//     PlcTask Inputs/MAIN.force_rb_X[146] <-> Status process data mapping/force_rb_X
//     PlcTask Inputs/MAIN.force_rb_Y[146] <-> Status process data mapping/force_rb_Y
//     PlcTask Inputs/MAIN.force_rb_Z[146] <-> Status process data mapping/force_rb_Z
//     PlcTask Inputs/MAIN.force_sp_X[146] <-> Status process data mapping/force_sp_X
//     PlcTask Inputs/MAIN.force_sp_Y[146] <-> Status process data mapping/force_sp_Y
//     PlcTask Inputs/MAIN.force_sp_Z[146] <-> Status process data mapping/force_sp_Z
//     PlcTask Inputs/MAIN.pwm1[146] <-> Status process data mapping/pwm1
//     PlcTask Inputs/MAIN.pwm2[146] <-> Status process data mapping/pwm2
//     PlcTask Inputs/MAIN.pwm3[146] <-> Status process data mapping/pwm3
//     PlcTask Outputs/MAIN.enable_cmd[146] <-> Control process data mapping/enable
//     PlcTask Outputs/MAIN.force_cmd_X[146] <-> Control process data mapping/force_sp_X
//     PlcTask Outputs/MAIN.force_cmd_Y[146] <-> Control process data mapping/force_sp_Y
//     PlcTask Outputs/MAIN.force_cmd_Z[146] <-> Control process data mapping/force_sp_Z
//     PlcTask Outputs/MAIN.msthb[156] <-> Control process data mapping/msthb
//   SAsetGains/SAsetGains Instance <-> Device 1 (EtherCAT)/Box 148 (m1eph)/Box 157 (m1sa)
//     PlcTask Inputs/MAIN.cloop_stat[147] <-> Status process data mapping/close_loop
//     PlcTask Inputs/MAIN.enable_stat[147] <-> Status process data mapping/enable
//     PlcTask Inputs/MAIN.force_rb_X[147] <-> Status process data mapping/force_rb_X
//     PlcTask Inputs/MAIN.force_rb_Y[147] <-> Status process data mapping/force_rb_Y
//     PlcTask Inputs/MAIN.force_rb_Z[147] <-> Status process data mapping/force_rb_Z
//     PlcTask Inputs/MAIN.force_sp_X[147] <-> Status process data mapping/force_sp_X
//     PlcTask Inputs/MAIN.force_sp_Y[147] <-> Status process data mapping/force_sp_Y
//     PlcTask Inputs/MAIN.force_sp_Z[147] <-> Status process data mapping/force_sp_Z
//     PlcTask Inputs/MAIN.pwm1[147] <-> Status process data mapping/pwm1
//     PlcTask Inputs/MAIN.pwm2[147] <-> Status process data mapping/pwm2
//     PlcTask Inputs/MAIN.pwm3[147] <-> Status process data mapping/pwm3
//     PlcTask Outputs/MAIN.enable_cmd[147] <-> Control process data mapping/enable
//     PlcTask Outputs/MAIN.force_cmd_X[147] <-> Control process data mapping/force_sp_X
//     PlcTask Outputs/MAIN.force_cmd_Y[147] <-> Control process data mapping/force_sp_Y
//     PlcTask Outputs/MAIN.force_cmd_Z[147] <-> Control process data mapping/force_sp_Z
//     PlcTask Outputs/MAIN.msthb[157] <-> Control process data mapping/msthb
//   SAsetGains/SAsetGains Instance <-> Device 1 (EtherCAT)/Box 148 (m1eph)/Box 158 (m1sa)
//     PlcTask Inputs/MAIN.cloop_stat[148] <-> Status process data mapping/close_loop
//     PlcTask Inputs/MAIN.enable_stat[148] <-> Status process data mapping/enable
//     PlcTask Inputs/MAIN.force_rb_X[148] <-> Status process data mapping/force_rb_X
//     PlcTask Inputs/MAIN.force_rb_Y[148] <-> Status process data mapping/force_rb_Y
//     PlcTask Inputs/MAIN.force_rb_Z[148] <-> Status process data mapping/force_rb_Z
//     PlcTask Inputs/MAIN.force_sp_X[148] <-> Status process data mapping/force_sp_X
//     PlcTask Inputs/MAIN.force_sp_Y[148] <-> Status process data mapping/force_sp_Y
//     PlcTask Inputs/MAIN.force_sp_Z[148] <-> Status process data mapping/force_sp_Z
//     PlcTask Inputs/MAIN.pwm1[148] <-> Status process data mapping/pwm1
//     PlcTask Inputs/MAIN.pwm2[148] <-> Status process data mapping/pwm2
//     PlcTask Inputs/MAIN.pwm3[148] <-> Status process data mapping/pwm3
//     PlcTask Outputs/MAIN.enable_cmd[148] <-> Control process data mapping/enable
//     PlcTask Outputs/MAIN.force_cmd_X[148] <-> Control process data mapping/force_sp_X
//     PlcTask Outputs/MAIN.force_cmd_Y[148] <-> Control process data mapping/force_sp_Y
//     PlcTask Outputs/MAIN.force_cmd_Z[148] <-> Control process data mapping/force_sp_Z
//     PlcTask Outputs/MAIN.msthb[158] <-> Control process data mapping/msthb
//   SAsetGains/SAsetGains Instance <-> Device 1 (EtherCAT)/Box 148 (m1eph)/Box 159 (m1sa)
//     PlcTask Inputs/MAIN.cloop_stat[149] <-> Status process data mapping/close_loop
//     PlcTask Inputs/MAIN.enable_stat[149] <-> Status process data mapping/enable
//     PlcTask Inputs/MAIN.force_rb_X[149] <-> Status process data mapping/force_rb_X
//     PlcTask Inputs/MAIN.force_rb_Y[149] <-> Status process data mapping/force_rb_Y
//     PlcTask Inputs/MAIN.force_rb_Z[149] <-> Status process data mapping/force_rb_Z
//     PlcTask Inputs/MAIN.force_sp_X[149] <-> Status process data mapping/force_sp_X
//     PlcTask Inputs/MAIN.force_sp_Y[149] <-> Status process data mapping/force_sp_Y
//     PlcTask Inputs/MAIN.force_sp_Z[149] <-> Status process data mapping/force_sp_Z
//     PlcTask Inputs/MAIN.pwm1[149] <-> Status process data mapping/pwm1
//     PlcTask Inputs/MAIN.pwm2[149] <-> Status process data mapping/pwm2
//     PlcTask Inputs/MAIN.pwm3[149] <-> Status process data mapping/pwm3
//     PlcTask Outputs/MAIN.enable_cmd[149] <-> Control process data mapping/enable
//     PlcTask Outputs/MAIN.force_cmd_X[149] <-> Control process data mapping/force_sp_X
//     PlcTask Outputs/MAIN.force_cmd_Y[149] <-> Control process data mapping/force_sp_Y
//     PlcTask Outputs/MAIN.force_cmd_Z[149] <-> Control process data mapping/force_sp_Z
//     PlcTask Outputs/MAIN.msthb[159] <-> Control process data mapping/msthb
//   SAsetGains/SAsetGains Instance <-> Device 1 (EtherCAT)/Box 148 (m1eph)/Box 160 (m1sa)
//     PlcTask Inputs/MAIN.cloop_stat[150] <-> Status process data mapping/close_loop
//     PlcTask Inputs/MAIN.enable_stat[150] <-> Status process data mapping/enable
//     PlcTask Inputs/MAIN.force_rb_X[150] <-> Status process data mapping/force_rb_X
//     PlcTask Inputs/MAIN.force_rb_Y[150] <-> Status process data mapping/force_rb_Y
//     PlcTask Inputs/MAIN.force_rb_Z[150] <-> Status process data mapping/force_rb_Z
//     PlcTask Inputs/MAIN.force_sp_X[150] <-> Status process data mapping/force_sp_X
//     PlcTask Inputs/MAIN.force_sp_Y[150] <-> Status process data mapping/force_sp_Y
//     PlcTask Inputs/MAIN.force_sp_Z[150] <-> Status process data mapping/force_sp_Z
//     PlcTask Inputs/MAIN.pwm1[150] <-> Status process data mapping/pwm1
//     PlcTask Inputs/MAIN.pwm2[150] <-> Status process data mapping/pwm2
//     PlcTask Inputs/MAIN.pwm3[150] <-> Status process data mapping/pwm3
//     PlcTask Outputs/MAIN.enable_cmd[150] <-> Control process data mapping/enable
//     PlcTask Outputs/MAIN.force_cmd_X[150] <-> Control process data mapping/force_sp_X
//     PlcTask Outputs/MAIN.force_cmd_Y[150] <-> Control process data mapping/force_sp_Y
//     PlcTask Outputs/MAIN.force_cmd_Z[150] <-> Control process data mapping/force_sp_Z
//     PlcTask Outputs/MAIN.msthb[160] <-> Control process data mapping/msthb
//   SAsetGains/SAsetGains Instance <-> Device 1 (EtherCAT)/Box 148 (m1eph)/Box 161 (m1sa)
//     PlcTask Inputs/MAIN.cloop_stat[151] <-> Status process data mapping/close_loop
//     PlcTask Inputs/MAIN.enable_stat[151] <-> Status process data mapping/enable
//     PlcTask Inputs/MAIN.force_rb_X[151] <-> Status process data mapping/force_rb_X
//     PlcTask Inputs/MAIN.force_rb_Y[151] <-> Status process data mapping/force_rb_Y
//     PlcTask Inputs/MAIN.force_rb_Z[151] <-> Status process data mapping/force_rb_Z
//     PlcTask Inputs/MAIN.force_sp_X[151] <-> Status process data mapping/force_sp_X
//     PlcTask Inputs/MAIN.force_sp_Y[151] <-> Status process data mapping/force_sp_Y
//     PlcTask Inputs/MAIN.force_sp_Z[151] <-> Status process data mapping/force_sp_Z
//     PlcTask Inputs/MAIN.pwm1[151] <-> Status process data mapping/pwm1
//     PlcTask Inputs/MAIN.pwm2[151] <-> Status process data mapping/pwm2
//     PlcTask Inputs/MAIN.pwm3[151] <-> Status process data mapping/pwm3
//     PlcTask Outputs/MAIN.enable_cmd[151] <-> Control process data mapping/enable
//     PlcTask Outputs/MAIN.force_cmd_X[151] <-> Control process data mapping/force_sp_X
//     PlcTask Outputs/MAIN.force_cmd_Y[151] <-> Control process data mapping/force_sp_Y
//     PlcTask Outputs/MAIN.force_cmd_Z[151] <-> Control process data mapping/force_sp_Z
//     PlcTask Outputs/MAIN.msthb[161] <-> Control process data mapping/msthb
//   SAsetGains/SAsetGains Instance <-> Device 1 (EtherCAT)/Box 148 (m1eph)/Box 162 (m1sa)
//     PlcTask Inputs/MAIN.cloop_stat[152] <-> Status process data mapping/close_loop
//     PlcTask Inputs/MAIN.enable_stat[152] <-> Status process data mapping/enable
//     PlcTask Inputs/MAIN.force_rb_X[152] <-> Status process data mapping/force_rb_X
//     PlcTask Inputs/MAIN.force_rb_Y[152] <-> Status process data mapping/force_rb_Y
//     PlcTask Inputs/MAIN.force_rb_Z[152] <-> Status process data mapping/force_rb_Z
//     PlcTask Inputs/MAIN.force_sp_X[152] <-> Status process data mapping/force_sp_X
//     PlcTask Inputs/MAIN.force_sp_Y[152] <-> Status process data mapping/force_sp_Y
//     PlcTask Inputs/MAIN.force_sp_Z[152] <-> Status process data mapping/force_sp_Z
//     PlcTask Inputs/MAIN.pwm1[152] <-> Status process data mapping/pwm1
//     PlcTask Inputs/MAIN.pwm2[152] <-> Status process data mapping/pwm2
//     PlcTask Inputs/MAIN.pwm3[152] <-> Status process data mapping/pwm3
//     PlcTask Outputs/MAIN.enable_cmd[152] <-> Control process data mapping/enable
//     PlcTask Outputs/MAIN.force_cmd_X[152] <-> Control process data mapping/force_sp_X
//     PlcTask Outputs/MAIN.force_cmd_Y[152] <-> Control process data mapping/force_sp_Y
//     PlcTask Outputs/MAIN.force_cmd_Z[152] <-> Control process data mapping/force_sp_Z
//     PlcTask Outputs/MAIN.msthb[162] <-> Control process data mapping/msthb
//   SAsetGains/SAsetGains Instance <-> Device 1 (EtherCAT)/Box 148 (m1eph)/Box 163 (m1sa)
//     PlcTask Inputs/MAIN.cloop_stat[153] <-> Status process data mapping/close_loop
//     PlcTask Inputs/MAIN.enable_stat[153] <-> Status process data mapping/enable
//     PlcTask Inputs/MAIN.force_rb_X[153] <-> Status process data mapping/force_rb_X
//     PlcTask Inputs/MAIN.force_rb_Y[153] <-> Status process data mapping/force_rb_Y
//     PlcTask Inputs/MAIN.force_rb_Z[153] <-> Status process data mapping/force_rb_Z
//     PlcTask Inputs/MAIN.force_sp_X[153] <-> Status process data mapping/force_sp_X
//     PlcTask Inputs/MAIN.force_sp_Y[153] <-> Status process data mapping/force_sp_Y
//     PlcTask Inputs/MAIN.force_sp_Z[153] <-> Status process data mapping/force_sp_Z
//     PlcTask Inputs/MAIN.pwm1[153] <-> Status process data mapping/pwm1
//     PlcTask Inputs/MAIN.pwm2[153] <-> Status process data mapping/pwm2
//     PlcTask Inputs/MAIN.pwm3[153] <-> Status process data mapping/pwm3
//     PlcTask Outputs/MAIN.enable_cmd[153] <-> Control process data mapping/enable
//     PlcTask Outputs/MAIN.force_cmd_X[153] <-> Control process data mapping/force_sp_X
//     PlcTask Outputs/MAIN.force_cmd_Y[153] <-> Control process data mapping/force_sp_Y
//     PlcTask Outputs/MAIN.force_cmd_Z[153] <-> Control process data mapping/force_sp_Z
//     PlcTask Outputs/MAIN.msthb[163] <-> Control process data mapping/msthb
//   SAsetGains/SAsetGains Instance <-> Device 1 (EtherCAT)/Box 148 (m1eph)/Box 164 (m1sa)
//     PlcTask Inputs/MAIN.cloop_stat[154] <-> Status process data mapping/close_loop
//     PlcTask Inputs/MAIN.enable_stat[154] <-> Status process data mapping/enable
//     PlcTask Inputs/MAIN.force_rb_X[154] <-> Status process data mapping/force_rb_X
//     PlcTask Inputs/MAIN.force_rb_Y[154] <-> Status process data mapping/force_rb_Y
//     PlcTask Inputs/MAIN.force_rb_Z[154] <-> Status process data mapping/force_rb_Z
//     PlcTask Inputs/MAIN.force_sp_X[154] <-> Status process data mapping/force_sp_X
//     PlcTask Inputs/MAIN.force_sp_Y[154] <-> Status process data mapping/force_sp_Y
//     PlcTask Inputs/MAIN.force_sp_Z[154] <-> Status process data mapping/force_sp_Z
//     PlcTask Inputs/MAIN.pwm1[154] <-> Status process data mapping/pwm1
//     PlcTask Inputs/MAIN.pwm2[154] <-> Status process data mapping/pwm2
//     PlcTask Inputs/MAIN.pwm3[154] <-> Status process data mapping/pwm3
//     PlcTask Outputs/MAIN.enable_cmd[154] <-> Control process data mapping/enable
//     PlcTask Outputs/MAIN.force_cmd_X[154] <-> Control process data mapping/force_sp_X
//     PlcTask Outputs/MAIN.force_cmd_Y[154] <-> Control process data mapping/force_sp_Y
//     PlcTask Outputs/MAIN.force_cmd_Z[154] <-> Control process data mapping/force_sp_Z
//     PlcTask Outputs/MAIN.msthb[164] <-> Control process data mapping/msthb
//   SAsetGains/SAsetGains Instance <-> Device 1 (EtherCAT)/Box 165 (m1eph)
//     PlcTask Outputs/MAIN.msthb[165] <-> Control process data mapping/msthb
//   SAsetGains/SAsetGains Instance <-> Device 1 (EtherCAT)/Box 165 (m1eph)/Box 166 (m1sa)
//     PlcTask Inputs/MAIN.cloop_stat[155] <-> Status process data mapping/close_loop
//     PlcTask Inputs/MAIN.enable_stat[155] <-> Status process data mapping/enable
//     PlcTask Inputs/MAIN.force_rb_X[155] <-> Status process data mapping/force_rb_X
//     PlcTask Inputs/MAIN.force_rb_Y[155] <-> Status process data mapping/force_rb_Y
//     PlcTask Inputs/MAIN.force_rb_Z[155] <-> Status process data mapping/force_rb_Z
//     PlcTask Inputs/MAIN.force_sp_X[155] <-> Status process data mapping/force_sp_X
//     PlcTask Inputs/MAIN.force_sp_Y[155] <-> Status process data mapping/force_sp_Y
//     PlcTask Inputs/MAIN.force_sp_Z[155] <-> Status process data mapping/force_sp_Z
//     PlcTask Inputs/MAIN.pwm1[155] <-> Status process data mapping/pwm1
//     PlcTask Inputs/MAIN.pwm2[155] <-> Status process data mapping/pwm2
//     PlcTask Inputs/MAIN.pwm3[155] <-> Status process data mapping/pwm3
//     PlcTask Outputs/MAIN.enable_cmd[155] <-> Control process data mapping/enable
//     PlcTask Outputs/MAIN.force_cmd_X[155] <-> Control process data mapping/force_sp_X
//     PlcTask Outputs/MAIN.force_cmd_Y[155] <-> Control process data mapping/force_sp_Y
//     PlcTask Outputs/MAIN.force_cmd_Z[155] <-> Control process data mapping/force_sp_Z
//     PlcTask Outputs/MAIN.msthb[166] <-> Control process data mapping/msthb
//   SAsetGains/SAsetGains Instance <-> Device 1 (EtherCAT)/Box 165 (m1eph)/Box 167 (m1sa)
//     PlcTask Inputs/MAIN.cloop_stat[156] <-> Status process data mapping/close_loop
//     PlcTask Inputs/MAIN.enable_stat[156] <-> Status process data mapping/enable
//     PlcTask Inputs/MAIN.force_rb_X[156] <-> Status process data mapping/force_rb_X
//     PlcTask Inputs/MAIN.force_rb_Y[156] <-> Status process data mapping/force_rb_Y
//     PlcTask Inputs/MAIN.force_rb_Z[156] <-> Status process data mapping/force_rb_Z
//     PlcTask Inputs/MAIN.force_sp_X[156] <-> Status process data mapping/force_sp_X
//     PlcTask Inputs/MAIN.force_sp_Y[156] <-> Status process data mapping/force_sp_Y
//     PlcTask Inputs/MAIN.force_sp_Z[156] <-> Status process data mapping/force_sp_Z
//     PlcTask Inputs/MAIN.pwm1[156] <-> Status process data mapping/pwm1
//     PlcTask Inputs/MAIN.pwm2[156] <-> Status process data mapping/pwm2
//     PlcTask Inputs/MAIN.pwm3[156] <-> Status process data mapping/pwm3
//     PlcTask Outputs/MAIN.enable_cmd[156] <-> Control process data mapping/enable
//     PlcTask Outputs/MAIN.force_cmd_X[156] <-> Control process data mapping/force_sp_X
//     PlcTask Outputs/MAIN.force_cmd_Y[156] <-> Control process data mapping/force_sp_Y
//     PlcTask Outputs/MAIN.force_cmd_Z[156] <-> Control process data mapping/force_sp_Z
//     PlcTask Outputs/MAIN.msthb[167] <-> Control process data mapping/msthb
//   SAsetGains/SAsetGains Instance <-> Device 1 (EtherCAT)/Box 165 (m1eph)/Box 168 (m1sa)
//     PlcTask Inputs/MAIN.cloop_stat[157] <-> Status process data mapping/close_loop
//     PlcTask Inputs/MAIN.enable_stat[157] <-> Status process data mapping/enable
//     PlcTask Inputs/MAIN.force_rb_X[157] <-> Status process data mapping/force_rb_X
//     PlcTask Inputs/MAIN.force_rb_Y[157] <-> Status process data mapping/force_rb_Y
//     PlcTask Inputs/MAIN.force_rb_Z[157] <-> Status process data mapping/force_rb_Z
//     PlcTask Inputs/MAIN.force_sp_X[157] <-> Status process data mapping/force_sp_X
//     PlcTask Inputs/MAIN.force_sp_Y[157] <-> Status process data mapping/force_sp_Y
//     PlcTask Inputs/MAIN.force_sp_Z[157] <-> Status process data mapping/force_sp_Z
//     PlcTask Inputs/MAIN.pwm1[157] <-> Status process data mapping/pwm1
//     PlcTask Inputs/MAIN.pwm2[157] <-> Status process data mapping/pwm2
//     PlcTask Inputs/MAIN.pwm3[157] <-> Status process data mapping/pwm3
//     PlcTask Outputs/MAIN.enable_cmd[157] <-> Control process data mapping/enable
//     PlcTask Outputs/MAIN.force_cmd_X[157] <-> Control process data mapping/force_sp_X
//     PlcTask Outputs/MAIN.force_cmd_Y[157] <-> Control process data mapping/force_sp_Y
//     PlcTask Outputs/MAIN.force_cmd_Z[157] <-> Control process data mapping/force_sp_Z
//     PlcTask Outputs/MAIN.msthb[168] <-> Control process data mapping/msthb
//   SAsetGains/SAsetGains Instance <-> Device 1 (EtherCAT)/Box 165 (m1eph)/Box 169 (m1sa)
//     PlcTask Inputs/MAIN.cloop_stat[158] <-> Status process data mapping/close_loop
//     PlcTask Inputs/MAIN.enable_stat[158] <-> Status process data mapping/enable
//     PlcTask Inputs/MAIN.force_rb_X[158] <-> Status process data mapping/force_rb_X
//     PlcTask Inputs/MAIN.force_rb_Y[158] <-> Status process data mapping/force_rb_Y
//     PlcTask Inputs/MAIN.force_rb_Z[158] <-> Status process data mapping/force_rb_Z
//     PlcTask Inputs/MAIN.force_sp_X[158] <-> Status process data mapping/force_sp_X
//     PlcTask Inputs/MAIN.force_sp_Y[158] <-> Status process data mapping/force_sp_Y
//     PlcTask Inputs/MAIN.force_sp_Z[158] <-> Status process data mapping/force_sp_Z
//     PlcTask Inputs/MAIN.pwm1[158] <-> Status process data mapping/pwm1
//     PlcTask Inputs/MAIN.pwm2[158] <-> Status process data mapping/pwm2
//     PlcTask Inputs/MAIN.pwm3[158] <-> Status process data mapping/pwm3
//     PlcTask Outputs/MAIN.enable_cmd[158] <-> Control process data mapping/enable
//     PlcTask Outputs/MAIN.force_cmd_X[158] <-> Control process data mapping/force_sp_X
//     PlcTask Outputs/MAIN.force_cmd_Y[158] <-> Control process data mapping/force_sp_Y
//     PlcTask Outputs/MAIN.force_cmd_Z[158] <-> Control process data mapping/force_sp_Z
//     PlcTask Outputs/MAIN.msthb[169] <-> Control process data mapping/msthb
//   SAsetGains/SAsetGains Instance <-> Device 1 (EtherCAT)/Box 165 (m1eph)/Box 170 (m1sa)
//     PlcTask Inputs/MAIN.cloop_stat[159] <-> Status process data mapping/close_loop
//     PlcTask Inputs/MAIN.enable_stat[159] <-> Status process data mapping/enable
//     PlcTask Inputs/MAIN.force_rb_X[159] <-> Status process data mapping/force_rb_X
//     PlcTask Inputs/MAIN.force_rb_Y[159] <-> Status process data mapping/force_rb_Y
//     PlcTask Inputs/MAIN.force_rb_Z[159] <-> Status process data mapping/force_rb_Z
//     PlcTask Inputs/MAIN.force_sp_X[159] <-> Status process data mapping/force_sp_X
//     PlcTask Inputs/MAIN.force_sp_Y[159] <-> Status process data mapping/force_sp_Y
//     PlcTask Inputs/MAIN.force_sp_Z[159] <-> Status process data mapping/force_sp_Z
//     PlcTask Inputs/MAIN.pwm1[159] <-> Status process data mapping/pwm1
//     PlcTask Inputs/MAIN.pwm2[159] <-> Status process data mapping/pwm2
//     PlcTask Inputs/MAIN.pwm3[159] <-> Status process data mapping/pwm3
//     PlcTask Outputs/MAIN.enable_cmd[159] <-> Control process data mapping/enable
//     PlcTask Outputs/MAIN.force_cmd_X[159] <-> Control process data mapping/force_sp_X
//     PlcTask Outputs/MAIN.force_cmd_Y[159] <-> Control process data mapping/force_sp_Y
//     PlcTask Outputs/MAIN.force_cmd_Z[159] <-> Control process data mapping/force_sp_Z
//     PlcTask Outputs/MAIN.msthb[170] <-> Control process data mapping/msthb
//   SAsetGains/SAsetGains Instance <-> Device 1 (EtherCAT)/Box 165 (m1eph)/Box 171 (m1sa)
//     PlcTask Inputs/MAIN.cloop_stat[160] <-> Status process data mapping/close_loop
//     PlcTask Inputs/MAIN.enable_stat[160] <-> Status process data mapping/enable
//     PlcTask Inputs/MAIN.force_rb_X[160] <-> Status process data mapping/force_rb_X
//     PlcTask Inputs/MAIN.force_rb_Y[160] <-> Status process data mapping/force_rb_Y
//     PlcTask Inputs/MAIN.force_rb_Z[160] <-> Status process data mapping/force_rb_Z
//     PlcTask Inputs/MAIN.force_sp_X[160] <-> Status process data mapping/force_sp_X
//     PlcTask Inputs/MAIN.force_sp_Y[160] <-> Status process data mapping/force_sp_Y
//     PlcTask Inputs/MAIN.force_sp_Z[160] <-> Status process data mapping/force_sp_Z
//     PlcTask Inputs/MAIN.pwm1[160] <-> Status process data mapping/pwm1
//     PlcTask Inputs/MAIN.pwm2[160] <-> Status process data mapping/pwm2
//     PlcTask Inputs/MAIN.pwm3[160] <-> Status process data mapping/pwm3
//     PlcTask Outputs/MAIN.enable_cmd[160] <-> Control process data mapping/enable
//     PlcTask Outputs/MAIN.force_cmd_X[160] <-> Control process data mapping/force_sp_X
//     PlcTask Outputs/MAIN.force_cmd_Y[160] <-> Control process data mapping/force_sp_Y
//     PlcTask Outputs/MAIN.force_cmd_Z[160] <-> Control process data mapping/force_sp_Z
//     PlcTask Outputs/MAIN.msthb[171] <-> Control process data mapping/msthb
//   SAsetGains/SAsetGains Instance <-> Device 1 (EtherCAT)/Box 165 (m1eph)/Box 172 (m1sa)
//     PlcTask Inputs/MAIN.cloop_stat[161] <-> Status process data mapping/close_loop
//     PlcTask Inputs/MAIN.enable_stat[161] <-> Status process data mapping/enable
//     PlcTask Inputs/MAIN.force_rb_X[161] <-> Status process data mapping/force_rb_X
//     PlcTask Inputs/MAIN.force_rb_Y[161] <-> Status process data mapping/force_rb_Y
//     PlcTask Inputs/MAIN.force_rb_Z[161] <-> Status process data mapping/force_rb_Z
//     PlcTask Inputs/MAIN.force_sp_X[161] <-> Status process data mapping/force_sp_X
//     PlcTask Inputs/MAIN.force_sp_Y[161] <-> Status process data mapping/force_sp_Y
//     PlcTask Inputs/MAIN.force_sp_Z[161] <-> Status process data mapping/force_sp_Z
//     PlcTask Inputs/MAIN.pwm1[161] <-> Status process data mapping/pwm1
//     PlcTask Inputs/MAIN.pwm2[161] <-> Status process data mapping/pwm2
//     PlcTask Inputs/MAIN.pwm3[161] <-> Status process data mapping/pwm3
//     PlcTask Outputs/MAIN.enable_cmd[161] <-> Control process data mapping/enable
//     PlcTask Outputs/MAIN.force_cmd_X[161] <-> Control process data mapping/force_sp_X
//     PlcTask Outputs/MAIN.force_cmd_Y[161] <-> Control process data mapping/force_sp_Y
//     PlcTask Outputs/MAIN.force_cmd_Z[161] <-> Control process data mapping/force_sp_Z
//     PlcTask Outputs/MAIN.msthb[172] <-> Control process data mapping/msthb
//   SAsetGains/SAsetGains Instance <-> Device 1 (EtherCAT)/Box 165 (m1eph)/Box 173 (m1sa)
//     PlcTask Inputs/MAIN.cloop_stat[162] <-> Status process data mapping/close_loop
//     PlcTask Inputs/MAIN.enable_stat[162] <-> Status process data mapping/enable
//     PlcTask Inputs/MAIN.force_rb_X[162] <-> Status process data mapping/force_rb_X
//     PlcTask Inputs/MAIN.force_rb_Y[162] <-> Status process data mapping/force_rb_Y
//     PlcTask Inputs/MAIN.force_rb_Z[162] <-> Status process data mapping/force_rb_Z
//     PlcTask Inputs/MAIN.force_sp_X[162] <-> Status process data mapping/force_sp_X
//     PlcTask Inputs/MAIN.force_sp_Y[162] <-> Status process data mapping/force_sp_Y
//     PlcTask Inputs/MAIN.force_sp_Z[162] <-> Status process data mapping/force_sp_Z
//     PlcTask Inputs/MAIN.pwm1[162] <-> Status process data mapping/pwm1
//     PlcTask Inputs/MAIN.pwm2[162] <-> Status process data mapping/pwm2
//     PlcTask Inputs/MAIN.pwm3[162] <-> Status process data mapping/pwm3
//     PlcTask Outputs/MAIN.enable_cmd[162] <-> Control process data mapping/enable
//     PlcTask Outputs/MAIN.force_cmd_X[162] <-> Control process data mapping/force_sp_X
//     PlcTask Outputs/MAIN.force_cmd_Y[162] <-> Control process data mapping/force_sp_Y
//     PlcTask Outputs/MAIN.force_cmd_Z[162] <-> Control process data mapping/force_sp_Z
//     PlcTask Outputs/MAIN.msthb[173] <-> Control process data mapping/msthb
//   SAsetGains/SAsetGains Instance <-> Device 1 (EtherCAT)/Box 165 (m1eph)/Box 174 (m1sa)
//     PlcTask Inputs/MAIN.cloop_stat[163] <-> Status process data mapping/close_loop
//     PlcTask Inputs/MAIN.enable_stat[163] <-> Status process data mapping/enable
//     PlcTask Inputs/MAIN.force_rb_X[163] <-> Status process data mapping/force_rb_X
//     PlcTask Inputs/MAIN.force_rb_Y[163] <-> Status process data mapping/force_rb_Y
//     PlcTask Inputs/MAIN.force_rb_Z[163] <-> Status process data mapping/force_rb_Z
//     PlcTask Inputs/MAIN.force_sp_X[163] <-> Status process data mapping/force_sp_X
//     PlcTask Inputs/MAIN.force_sp_Y[163] <-> Status process data mapping/force_sp_Y
//     PlcTask Inputs/MAIN.force_sp_Z[163] <-> Status process data mapping/force_sp_Z
//     PlcTask Inputs/MAIN.pwm1[163] <-> Status process data mapping/pwm1
//     PlcTask Inputs/MAIN.pwm2[163] <-> Status process data mapping/pwm2
//     PlcTask Inputs/MAIN.pwm3[163] <-> Status process data mapping/pwm3
//     PlcTask Outputs/MAIN.enable_cmd[163] <-> Control process data mapping/enable
//     PlcTask Outputs/MAIN.force_cmd_X[163] <-> Control process data mapping/force_sp_X
//     PlcTask Outputs/MAIN.force_cmd_Y[163] <-> Control process data mapping/force_sp_Y
//     PlcTask Outputs/MAIN.force_cmd_Z[163] <-> Control process data mapping/force_sp_Z
//     PlcTask Outputs/MAIN.msthb[174] <-> Control process data mapping/msthb
//   SAsetGains/SAsetGains Instance <-> Device 1 (EtherCAT)/Box 165 (m1eph)/Box 175 (m1sa)
//     PlcTask Inputs/MAIN.cloop_stat[164] <-> Status process data mapping/close_loop
//     PlcTask Inputs/MAIN.enable_stat[164] <-> Status process data mapping/enable
//     PlcTask Inputs/MAIN.force_rb_X[164] <-> Status process data mapping/force_rb_X
//     PlcTask Inputs/MAIN.force_rb_Y[164] <-> Status process data mapping/force_rb_Y
//     PlcTask Inputs/MAIN.force_rb_Z[164] <-> Status process data mapping/force_rb_Z
//     PlcTask Inputs/MAIN.force_sp_X[164] <-> Status process data mapping/force_sp_X
//     PlcTask Inputs/MAIN.force_sp_Y[164] <-> Status process data mapping/force_sp_Y
//     PlcTask Inputs/MAIN.force_sp_Z[164] <-> Status process data mapping/force_sp_Z
//     PlcTask Inputs/MAIN.pwm1[164] <-> Status process data mapping/pwm1
//     PlcTask Inputs/MAIN.pwm2[164] <-> Status process data mapping/pwm2
//     PlcTask Inputs/MAIN.pwm3[164] <-> Status process data mapping/pwm3
//     PlcTask Outputs/MAIN.enable_cmd[164] <-> Control process data mapping/enable
//     PlcTask Outputs/MAIN.force_cmd_X[164] <-> Control process data mapping/force_sp_X
//     PlcTask Outputs/MAIN.force_cmd_Y[164] <-> Control process data mapping/force_sp_Y
//     PlcTask Outputs/MAIN.force_cmd_Z[164] <-> Control process data mapping/force_sp_Z
//     PlcTask Outputs/MAIN.msthb[175] <-> Control process data mapping/msthb
//   SAsetGains/SAsetGains Instance <-> Device 1 (EtherCAT)/Box 165 (m1eph)/Box 176 (m1sa)
//     PlcTask Inputs/MAIN.cloop_stat[165] <-> Status process data mapping/close_loop
//     PlcTask Inputs/MAIN.enable_stat[165] <-> Status process data mapping/enable
//     PlcTask Inputs/MAIN.force_rb_X[165] <-> Status process data mapping/force_rb_X
//     PlcTask Inputs/MAIN.force_rb_Y[165] <-> Status process data mapping/force_rb_Y
//     PlcTask Inputs/MAIN.force_rb_Z[165] <-> Status process data mapping/force_rb_Z
//     PlcTask Inputs/MAIN.force_sp_X[165] <-> Status process data mapping/force_sp_X
//     PlcTask Inputs/MAIN.force_sp_Y[165] <-> Status process data mapping/force_sp_Y
//     PlcTask Inputs/MAIN.force_sp_Z[165] <-> Status process data mapping/force_sp_Z
//     PlcTask Inputs/MAIN.pwm1[165] <-> Status process data mapping/pwm1
//     PlcTask Inputs/MAIN.pwm2[165] <-> Status process data mapping/pwm2
//     PlcTask Inputs/MAIN.pwm3[165] <-> Status process data mapping/pwm3
//     PlcTask Outputs/MAIN.enable_cmd[165] <-> Control process data mapping/enable
//     PlcTask Outputs/MAIN.force_cmd_X[165] <-> Control process data mapping/force_sp_X
//     PlcTask Outputs/MAIN.force_cmd_Y[165] <-> Control process data mapping/force_sp_Y
//     PlcTask Outputs/MAIN.force_cmd_Z[165] <-> Control process data mapping/force_sp_Z
//     PlcTask Outputs/MAIN.msthb[176] <-> Control process data mapping/msthb
//   SAsetGains/SAsetGains Instance <-> Device 1 (EtherCAT)/Box 165 (m1eph)/Box 177 (m1sa)
//     PlcTask Inputs/MAIN.cloop_stat[166] <-> Status process data mapping/close_loop
//     PlcTask Inputs/MAIN.enable_stat[166] <-> Status process data mapping/enable
//     PlcTask Inputs/MAIN.force_rb_X[166] <-> Status process data mapping/force_rb_X
//     PlcTask Inputs/MAIN.force_rb_Y[166] <-> Status process data mapping/force_rb_Y
//     PlcTask Inputs/MAIN.force_rb_Z[166] <-> Status process data mapping/force_rb_Z
//     PlcTask Inputs/MAIN.force_sp_X[166] <-> Status process data mapping/force_sp_X
//     PlcTask Inputs/MAIN.force_sp_Y[166] <-> Status process data mapping/force_sp_Y
//     PlcTask Inputs/MAIN.force_sp_Z[166] <-> Status process data mapping/force_sp_Z
//     PlcTask Inputs/MAIN.pwm1[166] <-> Status process data mapping/pwm1
//     PlcTask Inputs/MAIN.pwm2[166] <-> Status process data mapping/pwm2
//     PlcTask Inputs/MAIN.pwm3[166] <-> Status process data mapping/pwm3
//     PlcTask Outputs/MAIN.enable_cmd[166] <-> Control process data mapping/enable
//     PlcTask Outputs/MAIN.force_cmd_X[166] <-> Control process data mapping/force_sp_X
//     PlcTask Outputs/MAIN.force_cmd_Y[166] <-> Control process data mapping/force_sp_Y
//     PlcTask Outputs/MAIN.force_cmd_Z[166] <-> Control process data mapping/force_sp_Z
//     PlcTask Outputs/MAIN.msthb[177] <-> Control process data mapping/msthb
//   SAsetGains/SAsetGains Instance <-> Device 1 (EtherCAT)/Box 165 (m1eph)/Box 178 (m1sa)
//     PlcTask Inputs/MAIN.cloop_stat[167] <-> Status process data mapping/close_loop
//     PlcTask Inputs/MAIN.enable_stat[167] <-> Status process data mapping/enable
//     PlcTask Inputs/MAIN.force_rb_X[167] <-> Status process data mapping/force_rb_X
//     PlcTask Inputs/MAIN.force_rb_Y[167] <-> Status process data mapping/force_rb_Y
//     PlcTask Inputs/MAIN.force_rb_Z[167] <-> Status process data mapping/force_rb_Z
//     PlcTask Inputs/MAIN.force_sp_X[167] <-> Status process data mapping/force_sp_X
//     PlcTask Inputs/MAIN.force_sp_Y[167] <-> Status process data mapping/force_sp_Y
//     PlcTask Inputs/MAIN.force_sp_Z[167] <-> Status process data mapping/force_sp_Z
//     PlcTask Inputs/MAIN.pwm1[167] <-> Status process data mapping/pwm1
//     PlcTask Inputs/MAIN.pwm2[167] <-> Status process data mapping/pwm2
//     PlcTask Inputs/MAIN.pwm3[167] <-> Status process data mapping/pwm3
//     PlcTask Outputs/MAIN.enable_cmd[167] <-> Control process data mapping/enable
//     PlcTask Outputs/MAIN.force_cmd_X[167] <-> Control process data mapping/force_sp_X
//     PlcTask Outputs/MAIN.force_cmd_Y[167] <-> Control process data mapping/force_sp_Y
//     PlcTask Outputs/MAIN.force_cmd_Z[167] <-> Control process data mapping/force_sp_Z
//     PlcTask Outputs/MAIN.msthb[178] <-> Control process data mapping/msthb
//   SAsetGains/SAsetGains Instance <-> Device 1 (EtherCAT)/Box 165 (m1eph)/Box 179 (m1sa)
//     PlcTask Inputs/MAIN.cloop_stat[168] <-> Status process data mapping/close_loop
//     PlcTask Inputs/MAIN.enable_stat[168] <-> Status process data mapping/enable
//     PlcTask Inputs/MAIN.force_rb_X[168] <-> Status process data mapping/force_rb_X
//     PlcTask Inputs/MAIN.force_rb_Y[168] <-> Status process data mapping/force_rb_Y
//     PlcTask Inputs/MAIN.force_rb_Z[168] <-> Status process data mapping/force_rb_Z
//     PlcTask Inputs/MAIN.force_sp_X[168] <-> Status process data mapping/force_sp_X
//     PlcTask Inputs/MAIN.force_sp_Y[168] <-> Status process data mapping/force_sp_Y
//     PlcTask Inputs/MAIN.force_sp_Z[168] <-> Status process data mapping/force_sp_Z
//     PlcTask Inputs/MAIN.pwm1[168] <-> Status process data mapping/pwm1
//     PlcTask Inputs/MAIN.pwm2[168] <-> Status process data mapping/pwm2
//     PlcTask Inputs/MAIN.pwm3[168] <-> Status process data mapping/pwm3
//     PlcTask Outputs/MAIN.enable_cmd[168] <-> Control process data mapping/enable
//     PlcTask Outputs/MAIN.force_cmd_X[168] <-> Control process data mapping/force_sp_X
//     PlcTask Outputs/MAIN.force_cmd_Y[168] <-> Control process data mapping/force_sp_Y
//     PlcTask Outputs/MAIN.force_cmd_Z[168] <-> Control process data mapping/force_sp_Z
//     PlcTask Outputs/MAIN.msthb[179] <-> Control process data mapping/msthb
//   SAsetGains/SAsetGains Instance <-> Device 1 (EtherCAT)/Box 165 (m1eph)/Box 180 (m1sa)
//     PlcTask Inputs/MAIN.cloop_stat[169] <-> Status process data mapping/close_loop
//     PlcTask Inputs/MAIN.enable_stat[169] <-> Status process data mapping/enable
//     PlcTask Inputs/MAIN.force_rb_X[169] <-> Status process data mapping/force_rb_X
//     PlcTask Inputs/MAIN.force_rb_Y[169] <-> Status process data mapping/force_rb_Y
//     PlcTask Inputs/MAIN.force_rb_Z[169] <-> Status process data mapping/force_rb_Z
//     PlcTask Inputs/MAIN.force_sp_X[169] <-> Status process data mapping/force_sp_X
//     PlcTask Inputs/MAIN.force_sp_Y[169] <-> Status process data mapping/force_sp_Y
//     PlcTask Inputs/MAIN.force_sp_Z[169] <-> Status process data mapping/force_sp_Z
//     PlcTask Inputs/MAIN.pwm1[169] <-> Status process data mapping/pwm1
//     PlcTask Inputs/MAIN.pwm2[169] <-> Status process data mapping/pwm2
//     PlcTask Inputs/MAIN.pwm3[169] <-> Status process data mapping/pwm3
//     PlcTask Outputs/MAIN.enable_cmd[169] <-> Control process data mapping/enable
//     PlcTask Outputs/MAIN.force_cmd_X[169] <-> Control process data mapping/force_sp_X
//     PlcTask Outputs/MAIN.force_cmd_Y[169] <-> Control process data mapping/force_sp_Y
//     PlcTask Outputs/MAIN.force_cmd_Z[169] <-> Control process data mapping/force_sp_Z
//     PlcTask Outputs/MAIN.msthb[180] <-> Control process data mapping/msthb
//   SAsetGains/SAsetGains Instance <-> Device 1 (EtherCAT)/Box 165 (m1eph)/Box 181 (m1sa)
//     PlcTask Inputs/MAIN.cloop_stat[170] <-> Status process data mapping/close_loop
//     PlcTask Inputs/MAIN.enable_stat[170] <-> Status process data mapping/enable
//     PlcTask Inputs/MAIN.force_rb_X[170] <-> Status process data mapping/force_rb_X
//     PlcTask Inputs/MAIN.force_rb_Y[170] <-> Status process data mapping/force_rb_Y
//     PlcTask Inputs/MAIN.force_rb_Z[170] <-> Status process data mapping/force_rb_Z
//     PlcTask Inputs/MAIN.force_sp_X[170] <-> Status process data mapping/force_sp_X
//     PlcTask Inputs/MAIN.force_sp_Y[170] <-> Status process data mapping/force_sp_Y
//     PlcTask Inputs/MAIN.force_sp_Z[170] <-> Status process data mapping/force_sp_Z
//     PlcTask Inputs/MAIN.pwm1[170] <-> Status process data mapping/pwm1
//     PlcTask Inputs/MAIN.pwm2[170] <-> Status process data mapping/pwm2
//     PlcTask Inputs/MAIN.pwm3[170] <-> Status process data mapping/pwm3
//     PlcTask Outputs/MAIN.enable_cmd[170] <-> Control process data mapping/enable
//     PlcTask Outputs/MAIN.force_cmd_X[170] <-> Control process data mapping/force_sp_X
//     PlcTask Outputs/MAIN.force_cmd_Y[170] <-> Control process data mapping/force_sp_Y
//     PlcTask Outputs/MAIN.force_cmd_Z[170] <-> Control process data mapping/force_sp_Z
//     PlcTask Outputs/MAIN.msthb[181] <-> Control process data mapping/msthb
//   SAsetGains/SAsetGains Instance <-> Device 1 (EtherCAT)/Box 18 (m1eph)
//     PlcTask Outputs/MAIN.msthb[18] <-> Control process data mapping/msthb
//   SAsetGains/SAsetGains Instance <-> Device 1 (EtherCAT)/Box 18 (m1eph)/Box 19 (m1sa)
//     PlcTask Inputs/MAIN.cloop_stat[17] <-> Status process data mapping/close_loop
//     PlcTask Inputs/MAIN.enable_stat[17] <-> Status process data mapping/enable
//     PlcTask Inputs/MAIN.force_rb_X[17] <-> Status process data mapping/force_rb_X
//     PlcTask Inputs/MAIN.force_rb_Y[17] <-> Status process data mapping/force_rb_Y
//     PlcTask Inputs/MAIN.force_rb_Z[17] <-> Status process data mapping/force_rb_Z
//     PlcTask Inputs/MAIN.force_sp_X[17] <-> Status process data mapping/force_sp_X
//     PlcTask Inputs/MAIN.force_sp_Y[17] <-> Status process data mapping/force_sp_Y
//     PlcTask Inputs/MAIN.force_sp_Z[17] <-> Status process data mapping/force_sp_Z
//     PlcTask Inputs/MAIN.pwm1[17] <-> Status process data mapping/pwm1
//     PlcTask Inputs/MAIN.pwm2[17] <-> Status process data mapping/pwm2
//     PlcTask Inputs/MAIN.pwm3[17] <-> Status process data mapping/pwm3
//     PlcTask Outputs/MAIN.enable_cmd[17] <-> Control process data mapping/enable
//     PlcTask Outputs/MAIN.force_cmd_X[17] <-> Control process data mapping/force_sp_X
//     PlcTask Outputs/MAIN.force_cmd_Y[17] <-> Control process data mapping/force_sp_Y
//     PlcTask Outputs/MAIN.force_cmd_Z[17] <-> Control process data mapping/force_sp_Z
//     PlcTask Outputs/MAIN.msthb[19] <-> Control process data mapping/msthb
//   SAsetGains/SAsetGains Instance <-> Device 1 (EtherCAT)/Box 18 (m1eph)/Box 20 (m1sa)
//     PlcTask Inputs/MAIN.cloop_stat[18] <-> Status process data mapping/close_loop
//     PlcTask Inputs/MAIN.enable_stat[18] <-> Status process data mapping/enable
//     PlcTask Inputs/MAIN.force_rb_X[18] <-> Status process data mapping/force_rb_X
//     PlcTask Inputs/MAIN.force_rb_Y[18] <-> Status process data mapping/force_rb_Y
//     PlcTask Inputs/MAIN.force_rb_Z[18] <-> Status process data mapping/force_rb_Z
//     PlcTask Inputs/MAIN.force_sp_X[18] <-> Status process data mapping/force_sp_X
//     PlcTask Inputs/MAIN.force_sp_Y[18] <-> Status process data mapping/force_sp_Y
//     PlcTask Inputs/MAIN.force_sp_Z[18] <-> Status process data mapping/force_sp_Z
//     PlcTask Inputs/MAIN.pwm1[18] <-> Status process data mapping/pwm1
//     PlcTask Inputs/MAIN.pwm2[18] <-> Status process data mapping/pwm2
//     PlcTask Inputs/MAIN.pwm3[18] <-> Status process data mapping/pwm3
//     PlcTask Outputs/MAIN.enable_cmd[18] <-> Control process data mapping/enable
//     PlcTask Outputs/MAIN.force_cmd_X[18] <-> Control process data mapping/force_sp_X
//     PlcTask Outputs/MAIN.force_cmd_Y[18] <-> Control process data mapping/force_sp_Y
//     PlcTask Outputs/MAIN.force_cmd_Z[18] <-> Control process data mapping/force_sp_Z
//     PlcTask Outputs/MAIN.msthb[20] <-> Control process data mapping/msthb
//   SAsetGains/SAsetGains Instance <-> Device 1 (EtherCAT)/Box 18 (m1eph)/Box 21 (m1sa)
//     PlcTask Inputs/MAIN.cloop_stat[19] <-> Status process data mapping/close_loop
//     PlcTask Inputs/MAIN.enable_stat[19] <-> Status process data mapping/enable
//     PlcTask Inputs/MAIN.force_rb_X[19] <-> Status process data mapping/force_rb_X
//     PlcTask Inputs/MAIN.force_rb_Y[19] <-> Status process data mapping/force_rb_Y
//     PlcTask Inputs/MAIN.force_rb_Z[19] <-> Status process data mapping/force_rb_Z
//     PlcTask Inputs/MAIN.force_sp_X[19] <-> Status process data mapping/force_sp_X
//     PlcTask Inputs/MAIN.force_sp_Y[19] <-> Status process data mapping/force_sp_Y
//     PlcTask Inputs/MAIN.force_sp_Z[19] <-> Status process data mapping/force_sp_Z
//     PlcTask Inputs/MAIN.pwm1[19] <-> Status process data mapping/pwm1
//     PlcTask Inputs/MAIN.pwm2[19] <-> Status process data mapping/pwm2
//     PlcTask Inputs/MAIN.pwm3[19] <-> Status process data mapping/pwm3
//     PlcTask Outputs/MAIN.enable_cmd[19] <-> Control process data mapping/enable
//     PlcTask Outputs/MAIN.force_cmd_X[19] <-> Control process data mapping/force_sp_X
//     PlcTask Outputs/MAIN.force_cmd_Y[19] <-> Control process data mapping/force_sp_Y
//     PlcTask Outputs/MAIN.force_cmd_Z[19] <-> Control process data mapping/force_sp_Z
//     PlcTask Outputs/MAIN.msthb[21] <-> Control process data mapping/msthb
//   SAsetGains/SAsetGains Instance <-> Device 1 (EtherCAT)/Box 18 (m1eph)/Box 22 (m1sa)
//     PlcTask Inputs/MAIN.cloop_stat[20] <-> Status process data mapping/close_loop
//     PlcTask Inputs/MAIN.enable_stat[20] <-> Status process data mapping/enable
//     PlcTask Inputs/MAIN.force_rb_X[20] <-> Status process data mapping/force_rb_X
//     PlcTask Inputs/MAIN.force_rb_Y[20] <-> Status process data mapping/force_rb_Y
//     PlcTask Inputs/MAIN.force_rb_Z[20] <-> Status process data mapping/force_rb_Z
//     PlcTask Inputs/MAIN.force_sp_X[20] <-> Status process data mapping/force_sp_X
//     PlcTask Inputs/MAIN.force_sp_Y[20] <-> Status process data mapping/force_sp_Y
//     PlcTask Inputs/MAIN.force_sp_Z[20] <-> Status process data mapping/force_sp_Z
//     PlcTask Inputs/MAIN.pwm1[20] <-> Status process data mapping/pwm1
//     PlcTask Inputs/MAIN.pwm2[20] <-> Status process data mapping/pwm2
//     PlcTask Inputs/MAIN.pwm3[20] <-> Status process data mapping/pwm3
//     PlcTask Outputs/MAIN.enable_cmd[20] <-> Control process data mapping/enable
//     PlcTask Outputs/MAIN.force_cmd_X[20] <-> Control process data mapping/force_sp_X
//     PlcTask Outputs/MAIN.force_cmd_Y[20] <-> Control process data mapping/force_sp_Y
//     PlcTask Outputs/MAIN.force_cmd_Z[20] <-> Control process data mapping/force_sp_Z
//     PlcTask Outputs/MAIN.msthb[22] <-> Control process data mapping/msthb
//   SAsetGains/SAsetGains Instance <-> Device 1 (EtherCAT)/Box 18 (m1eph)/Box 23 (m1sa)
//     PlcTask Inputs/MAIN.cloop_stat[21] <-> Status process data mapping/close_loop
//     PlcTask Inputs/MAIN.enable_stat[21] <-> Status process data mapping/enable
//     PlcTask Inputs/MAIN.force_rb_X[21] <-> Status process data mapping/force_rb_X
//     PlcTask Inputs/MAIN.force_rb_Y[21] <-> Status process data mapping/force_rb_Y
//     PlcTask Inputs/MAIN.force_rb_Z[21] <-> Status process data mapping/force_rb_Z
//     PlcTask Inputs/MAIN.force_sp_X[21] <-> Status process data mapping/force_sp_X
//     PlcTask Inputs/MAIN.force_sp_Y[21] <-> Status process data mapping/force_sp_Y
//     PlcTask Inputs/MAIN.force_sp_Z[21] <-> Status process data mapping/force_sp_Z
//     PlcTask Inputs/MAIN.pwm1[21] <-> Status process data mapping/pwm1
//     PlcTask Inputs/MAIN.pwm2[21] <-> Status process data mapping/pwm2
//     PlcTask Inputs/MAIN.pwm3[21] <-> Status process data mapping/pwm3
//     PlcTask Outputs/MAIN.enable_cmd[21] <-> Control process data mapping/enable
//     PlcTask Outputs/MAIN.force_cmd_X[21] <-> Control process data mapping/force_sp_X
//     PlcTask Outputs/MAIN.force_cmd_Y[21] <-> Control process data mapping/force_sp_Y
//     PlcTask Outputs/MAIN.force_cmd_Z[21] <-> Control process data mapping/force_sp_Z
//     PlcTask Outputs/MAIN.msthb[23] <-> Control process data mapping/msthb
//   SAsetGains/SAsetGains Instance <-> Device 1 (EtherCAT)/Box 18 (m1eph)/Box 24 (m1sa)
//     PlcTask Inputs/MAIN.cloop_stat[22] <-> Status process data mapping/close_loop
//     PlcTask Inputs/MAIN.enable_stat[22] <-> Status process data mapping/enable
//     PlcTask Inputs/MAIN.force_rb_X[22] <-> Status process data mapping/force_rb_X
//     PlcTask Inputs/MAIN.force_rb_Y[22] <-> Status process data mapping/force_rb_Y
//     PlcTask Inputs/MAIN.force_rb_Z[22] <-> Status process data mapping/force_rb_Z
//     PlcTask Inputs/MAIN.force_sp_X[22] <-> Status process data mapping/force_sp_X
//     PlcTask Inputs/MAIN.force_sp_Y[22] <-> Status process data mapping/force_sp_Y
//     PlcTask Inputs/MAIN.force_sp_Z[22] <-> Status process data mapping/force_sp_Z
//     PlcTask Inputs/MAIN.pwm1[22] <-> Status process data mapping/pwm1
//     PlcTask Inputs/MAIN.pwm2[22] <-> Status process data mapping/pwm2
//     PlcTask Inputs/MAIN.pwm3[22] <-> Status process data mapping/pwm3
//     PlcTask Outputs/MAIN.enable_cmd[22] <-> Control process data mapping/enable
//     PlcTask Outputs/MAIN.force_cmd_X[22] <-> Control process data mapping/force_sp_X
//     PlcTask Outputs/MAIN.force_cmd_Y[22] <-> Control process data mapping/force_sp_Y
//     PlcTask Outputs/MAIN.force_cmd_Z[22] <-> Control process data mapping/force_sp_Z
//     PlcTask Outputs/MAIN.msthb[24] <-> Control process data mapping/msthb
//   SAsetGains/SAsetGains Instance <-> Device 1 (EtherCAT)/Box 18 (m1eph)/Box 25 (m1sa)
//     PlcTask Inputs/MAIN.cloop_stat[23] <-> Status process data mapping/close_loop
//     PlcTask Inputs/MAIN.enable_stat[23] <-> Status process data mapping/enable
//     PlcTask Inputs/MAIN.force_rb_X[23] <-> Status process data mapping/force_rb_X
//     PlcTask Inputs/MAIN.force_rb_Y[23] <-> Status process data mapping/force_rb_Y
//     PlcTask Inputs/MAIN.force_rb_Z[23] <-> Status process data mapping/force_rb_Z
//     PlcTask Inputs/MAIN.force_sp_X[23] <-> Status process data mapping/force_sp_X
//     PlcTask Inputs/MAIN.force_sp_Y[23] <-> Status process data mapping/force_sp_Y
//     PlcTask Inputs/MAIN.force_sp_Z[23] <-> Status process data mapping/force_sp_Z
//     PlcTask Inputs/MAIN.pwm1[23] <-> Status process data mapping/pwm1
//     PlcTask Inputs/MAIN.pwm2[23] <-> Status process data mapping/pwm2
//     PlcTask Inputs/MAIN.pwm3[23] <-> Status process data mapping/pwm3
//     PlcTask Outputs/MAIN.enable_cmd[23] <-> Control process data mapping/enable
//     PlcTask Outputs/MAIN.force_cmd_X[23] <-> Control process data mapping/force_sp_X
//     PlcTask Outputs/MAIN.force_cmd_Y[23] <-> Control process data mapping/force_sp_Y
//     PlcTask Outputs/MAIN.force_cmd_Z[23] <-> Control process data mapping/force_sp_Z
//     PlcTask Outputs/MAIN.msthb[25] <-> Control process data mapping/msthb
//   SAsetGains/SAsetGains Instance <-> Device 1 (EtherCAT)/Box 18 (m1eph)/Box 26 (m1sa)
//     PlcTask Inputs/MAIN.cloop_stat[24] <-> Status process data mapping/close_loop
//     PlcTask Inputs/MAIN.enable_stat[24] <-> Status process data mapping/enable
//     PlcTask Inputs/MAIN.force_rb_X[24] <-> Status process data mapping/force_rb_X
//     PlcTask Inputs/MAIN.force_rb_Y[24] <-> Status process data mapping/force_rb_Y
//     PlcTask Inputs/MAIN.force_rb_Z[24] <-> Status process data mapping/force_rb_Z
//     PlcTask Inputs/MAIN.force_sp_X[24] <-> Status process data mapping/force_sp_X
//     PlcTask Inputs/MAIN.force_sp_Y[24] <-> Status process data mapping/force_sp_Y
//     PlcTask Inputs/MAIN.force_sp_Z[24] <-> Status process data mapping/force_sp_Z
//     PlcTask Inputs/MAIN.pwm1[24] <-> Status process data mapping/pwm1
//     PlcTask Inputs/MAIN.pwm2[24] <-> Status process data mapping/pwm2
//     PlcTask Inputs/MAIN.pwm3[24] <-> Status process data mapping/pwm3
//     PlcTask Outputs/MAIN.enable_cmd[24] <-> Control process data mapping/enable
//     PlcTask Outputs/MAIN.force_cmd_X[24] <-> Control process data mapping/force_sp_X
//     PlcTask Outputs/MAIN.force_cmd_Y[24] <-> Control process data mapping/force_sp_Y
//     PlcTask Outputs/MAIN.force_cmd_Z[24] <-> Control process data mapping/force_sp_Z
//     PlcTask Outputs/MAIN.msthb[26] <-> Control process data mapping/msthb
//   SAsetGains/SAsetGains Instance <-> Device 1 (EtherCAT)/Box 18 (m1eph)/Box 27 (m1sa)
//     PlcTask Inputs/MAIN.cloop_stat[25] <-> Status process data mapping/close_loop
//     PlcTask Inputs/MAIN.enable_stat[25] <-> Status process data mapping/enable
//     PlcTask Inputs/MAIN.force_rb_X[25] <-> Status process data mapping/force_rb_X
//     PlcTask Inputs/MAIN.force_rb_Y[25] <-> Status process data mapping/force_rb_Y
//     PlcTask Inputs/MAIN.force_rb_Z[25] <-> Status process data mapping/force_rb_Z
//     PlcTask Inputs/MAIN.force_sp_X[25] <-> Status process data mapping/force_sp_X
//     PlcTask Inputs/MAIN.force_sp_Y[25] <-> Status process data mapping/force_sp_Y
//     PlcTask Inputs/MAIN.force_sp_Z[25] <-> Status process data mapping/force_sp_Z
//     PlcTask Inputs/MAIN.pwm1[25] <-> Status process data mapping/pwm1
//     PlcTask Inputs/MAIN.pwm2[25] <-> Status process data mapping/pwm2
//     PlcTask Inputs/MAIN.pwm3[25] <-> Status process data mapping/pwm3
//     PlcTask Outputs/MAIN.enable_cmd[25] <-> Control process data mapping/enable
//     PlcTask Outputs/MAIN.force_cmd_X[25] <-> Control process data mapping/force_sp_X
//     PlcTask Outputs/MAIN.force_cmd_Y[25] <-> Control process data mapping/force_sp_Y
//     PlcTask Outputs/MAIN.force_cmd_Z[25] <-> Control process data mapping/force_sp_Z
//     PlcTask Outputs/MAIN.msthb[27] <-> Control process data mapping/msthb
//   SAsetGains/SAsetGains Instance <-> Device 1 (EtherCAT)/Box 18 (m1eph)/Box 28 (m1sa)
//     PlcTask Inputs/MAIN.cloop_stat[26] <-> Status process data mapping/close_loop
//     PlcTask Inputs/MAIN.enable_stat[26] <-> Status process data mapping/enable
//     PlcTask Inputs/MAIN.force_rb_X[26] <-> Status process data mapping/force_rb_X
//     PlcTask Inputs/MAIN.force_rb_Y[26] <-> Status process data mapping/force_rb_Y
//     PlcTask Inputs/MAIN.force_rb_Z[26] <-> Status process data mapping/force_rb_Z
//     PlcTask Inputs/MAIN.force_sp_X[26] <-> Status process data mapping/force_sp_X
//     PlcTask Inputs/MAIN.force_sp_Y[26] <-> Status process data mapping/force_sp_Y
//     PlcTask Inputs/MAIN.force_sp_Z[26] <-> Status process data mapping/force_sp_Z
//     PlcTask Inputs/MAIN.pwm1[26] <-> Status process data mapping/pwm1
//     PlcTask Inputs/MAIN.pwm2[26] <-> Status process data mapping/pwm2
//     PlcTask Inputs/MAIN.pwm3[26] <-> Status process data mapping/pwm3
//     PlcTask Outputs/MAIN.enable_cmd[26] <-> Control process data mapping/enable
//     PlcTask Outputs/MAIN.force_cmd_X[26] <-> Control process data mapping/force_sp_X
//     PlcTask Outputs/MAIN.force_cmd_Y[26] <-> Control process data mapping/force_sp_Y
//     PlcTask Outputs/MAIN.force_cmd_Z[26] <-> Control process data mapping/force_sp_Z
//     PlcTask Outputs/MAIN.msthb[28] <-> Control process data mapping/msthb
//   SAsetGains/SAsetGains Instance <-> Device 1 (EtherCAT)/Box 18 (m1eph)/Box 29 (m1sa)
//     PlcTask Inputs/MAIN.cloop_stat[27] <-> Status process data mapping/close_loop
//     PlcTask Inputs/MAIN.enable_stat[27] <-> Status process data mapping/enable
//     PlcTask Inputs/MAIN.force_rb_X[27] <-> Status process data mapping/force_rb_X
//     PlcTask Inputs/MAIN.force_rb_Y[27] <-> Status process data mapping/force_rb_Y
//     PlcTask Inputs/MAIN.force_rb_Z[27] <-> Status process data mapping/force_rb_Z
//     PlcTask Inputs/MAIN.force_sp_X[27] <-> Status process data mapping/force_sp_X
//     PlcTask Inputs/MAIN.force_sp_Y[27] <-> Status process data mapping/force_sp_Y
//     PlcTask Inputs/MAIN.force_sp_Z[27] <-> Status process data mapping/force_sp_Z
//     PlcTask Inputs/MAIN.pwm1[27] <-> Status process data mapping/pwm1
//     PlcTask Inputs/MAIN.pwm2[27] <-> Status process data mapping/pwm2
//     PlcTask Inputs/MAIN.pwm3[27] <-> Status process data mapping/pwm3
//     PlcTask Outputs/MAIN.enable_cmd[27] <-> Control process data mapping/enable
//     PlcTask Outputs/MAIN.force_cmd_X[27] <-> Control process data mapping/force_sp_X
//     PlcTask Outputs/MAIN.force_cmd_Y[27] <-> Control process data mapping/force_sp_Y
//     PlcTask Outputs/MAIN.force_cmd_Z[27] <-> Control process data mapping/force_sp_Z
//     PlcTask Outputs/MAIN.msthb[29] <-> Control process data mapping/msthb
//   SAsetGains/SAsetGains Instance <-> Device 1 (EtherCAT)/Box 18 (m1eph)/Box 30 (m1sa)
//     PlcTask Inputs/MAIN.cloop_stat[28] <-> Status process data mapping/close_loop
//     PlcTask Inputs/MAIN.enable_stat[28] <-> Status process data mapping/enable
//     PlcTask Inputs/MAIN.force_rb_X[28] <-> Status process data mapping/force_rb_X
//     PlcTask Inputs/MAIN.force_rb_Y[28] <-> Status process data mapping/force_rb_Y
//     PlcTask Inputs/MAIN.force_rb_Z[28] <-> Status process data mapping/force_rb_Z
//     PlcTask Inputs/MAIN.force_sp_X[28] <-> Status process data mapping/force_sp_X
//     PlcTask Inputs/MAIN.force_sp_Y[28] <-> Status process data mapping/force_sp_Y
//     PlcTask Inputs/MAIN.force_sp_Z[28] <-> Status process data mapping/force_sp_Z
//     PlcTask Inputs/MAIN.pwm1[28] <-> Status process data mapping/pwm1
//     PlcTask Inputs/MAIN.pwm2[28] <-> Status process data mapping/pwm2
//     PlcTask Inputs/MAIN.pwm3[28] <-> Status process data mapping/pwm3
//     PlcTask Outputs/MAIN.enable_cmd[28] <-> Control process data mapping/enable
//     PlcTask Outputs/MAIN.force_cmd_X[28] <-> Control process data mapping/force_sp_X
//     PlcTask Outputs/MAIN.force_cmd_Y[28] <-> Control process data mapping/force_sp_Y
//     PlcTask Outputs/MAIN.force_cmd_Z[28] <-> Control process data mapping/force_sp_Z
//     PlcTask Outputs/MAIN.msthb[30] <-> Control process data mapping/msthb
//   SAsetGains/SAsetGains Instance <-> Device 1 (EtherCAT)/Box 18 (m1eph)/Box 31 (m1sa)
//     PlcTask Inputs/MAIN.cloop_stat[29] <-> Status process data mapping/close_loop
//     PlcTask Inputs/MAIN.enable_stat[29] <-> Status process data mapping/enable
//     PlcTask Inputs/MAIN.force_rb_X[29] <-> Status process data mapping/force_rb_X
//     PlcTask Inputs/MAIN.force_rb_Y[29] <-> Status process data mapping/force_rb_Y
//     PlcTask Inputs/MAIN.force_rb_Z[29] <-> Status process data mapping/force_rb_Z
//     PlcTask Inputs/MAIN.force_sp_X[29] <-> Status process data mapping/force_sp_X
//     PlcTask Inputs/MAIN.force_sp_Y[29] <-> Status process data mapping/force_sp_Y
//     PlcTask Inputs/MAIN.force_sp_Z[29] <-> Status process data mapping/force_sp_Z
//     PlcTask Inputs/MAIN.pwm1[29] <-> Status process data mapping/pwm1
//     PlcTask Inputs/MAIN.pwm2[29] <-> Status process data mapping/pwm2
//     PlcTask Inputs/MAIN.pwm3[29] <-> Status process data mapping/pwm3
//     PlcTask Outputs/MAIN.enable_cmd[29] <-> Control process data mapping/enable
//     PlcTask Outputs/MAIN.force_cmd_X[29] <-> Control process data mapping/force_sp_X
//     PlcTask Outputs/MAIN.force_cmd_Y[29] <-> Control process data mapping/force_sp_Y
//     PlcTask Outputs/MAIN.force_cmd_Z[29] <-> Control process data mapping/force_sp_Z
//     PlcTask Outputs/MAIN.msthb[31] <-> Control process data mapping/msthb
//   SAsetGains/SAsetGains Instance <-> Device 1 (EtherCAT)/Box 18 (m1eph)/Box 32 (m1sa)
//     PlcTask Inputs/MAIN.cloop_stat[30] <-> Status process data mapping/close_loop
//     PlcTask Inputs/MAIN.enable_stat[30] <-> Status process data mapping/enable
//     PlcTask Inputs/MAIN.force_rb_X[30] <-> Status process data mapping/force_rb_X
//     PlcTask Inputs/MAIN.force_rb_Y[30] <-> Status process data mapping/force_rb_Y
//     PlcTask Inputs/MAIN.force_rb_Z[30] <-> Status process data mapping/force_rb_Z
//     PlcTask Inputs/MAIN.force_sp_X[30] <-> Status process data mapping/force_sp_X
//     PlcTask Inputs/MAIN.force_sp_Y[30] <-> Status process data mapping/force_sp_Y
//     PlcTask Inputs/MAIN.force_sp_Z[30] <-> Status process data mapping/force_sp_Z
//     PlcTask Inputs/MAIN.pwm1[30] <-> Status process data mapping/pwm1
//     PlcTask Inputs/MAIN.pwm2[30] <-> Status process data mapping/pwm2
//     PlcTask Inputs/MAIN.pwm3[30] <-> Status process data mapping/pwm3
//     PlcTask Outputs/MAIN.enable_cmd[30] <-> Control process data mapping/enable
//     PlcTask Outputs/MAIN.force_cmd_X[30] <-> Control process data mapping/force_sp_X
//     PlcTask Outputs/MAIN.force_cmd_Y[30] <-> Control process data mapping/force_sp_Y
//     PlcTask Outputs/MAIN.force_cmd_Z[30] <-> Control process data mapping/force_sp_Z
//     PlcTask Outputs/MAIN.msthb[32] <-> Control process data mapping/msthb
//   SAsetGains/SAsetGains Instance <-> Device 1 (EtherCAT)/Box 33 (m1eph)
//     PlcTask Outputs/MAIN.msthb[33] <-> Control process data mapping/msthb
//   SAsetGains/SAsetGains Instance <-> Device 1 (EtherCAT)/Box 33 (m1eph)/Box 34 (m1sa)
//     PlcTask Inputs/MAIN.cloop_stat[31] <-> Status process data mapping/close_loop
//     PlcTask Inputs/MAIN.enable_stat[31] <-> Status process data mapping/enable
//     PlcTask Inputs/MAIN.force_rb_X[31] <-> Status process data mapping/force_rb_X
//     PlcTask Inputs/MAIN.force_rb_Y[31] <-> Status process data mapping/force_rb_Y
//     PlcTask Inputs/MAIN.force_rb_Z[31] <-> Status process data mapping/force_rb_Z
//     PlcTask Inputs/MAIN.force_sp_X[31] <-> Status process data mapping/force_sp_X
//     PlcTask Inputs/MAIN.force_sp_Y[31] <-> Status process data mapping/force_sp_Y
//     PlcTask Inputs/MAIN.force_sp_Z[31] <-> Status process data mapping/force_sp_Z
//     PlcTask Inputs/MAIN.pwm1[31] <-> Status process data mapping/pwm1
//     PlcTask Inputs/MAIN.pwm2[31] <-> Status process data mapping/pwm2
//     PlcTask Inputs/MAIN.pwm3[31] <-> Status process data mapping/pwm3
//     PlcTask Outputs/MAIN.enable_cmd[31] <-> Control process data mapping/enable
//     PlcTask Outputs/MAIN.force_cmd_X[31] <-> Control process data mapping/force_sp_X
//     PlcTask Outputs/MAIN.force_cmd_Y[31] <-> Control process data mapping/force_sp_Y
//     PlcTask Outputs/MAIN.force_cmd_Z[31] <-> Control process data mapping/force_sp_Z
//     PlcTask Outputs/MAIN.msthb[34] <-> Control process data mapping/msthb
//   SAsetGains/SAsetGains Instance <-> Device 1 (EtherCAT)/Box 33 (m1eph)/Box 35 (m1sa)
//     PlcTask Inputs/MAIN.cloop_stat[32] <-> Status process data mapping/close_loop
//     PlcTask Inputs/MAIN.enable_stat[32] <-> Status process data mapping/enable
//     PlcTask Inputs/MAIN.force_rb_X[32] <-> Status process data mapping/force_rb_X
//     PlcTask Inputs/MAIN.force_rb_Y[32] <-> Status process data mapping/force_rb_Y
//     PlcTask Inputs/MAIN.force_rb_Z[32] <-> Status process data mapping/force_rb_Z
//     PlcTask Inputs/MAIN.force_sp_X[32] <-> Status process data mapping/force_sp_X
//     PlcTask Inputs/MAIN.force_sp_Y[32] <-> Status process data mapping/force_sp_Y
//     PlcTask Inputs/MAIN.force_sp_Z[32] <-> Status process data mapping/force_sp_Z
//     PlcTask Inputs/MAIN.pwm1[32] <-> Status process data mapping/pwm1
//     PlcTask Inputs/MAIN.pwm2[32] <-> Status process data mapping/pwm2
//     PlcTask Inputs/MAIN.pwm3[32] <-> Status process data mapping/pwm3
//     PlcTask Outputs/MAIN.enable_cmd[32] <-> Control process data mapping/enable
//     PlcTask Outputs/MAIN.force_cmd_X[32] <-> Control process data mapping/force_sp_X
//     PlcTask Outputs/MAIN.force_cmd_Y[32] <-> Control process data mapping/force_sp_Y
//     PlcTask Outputs/MAIN.force_cmd_Z[32] <-> Control process data mapping/force_sp_Z
//     PlcTask Outputs/MAIN.msthb[35] <-> Control process data mapping/msthb
//   SAsetGains/SAsetGains Instance <-> Device 1 (EtherCAT)/Box 33 (m1eph)/Box 36 (m1sa)
//     PlcTask Inputs/MAIN.cloop_stat[33] <-> Status process data mapping/close_loop
//     PlcTask Inputs/MAIN.enable_stat[33] <-> Status process data mapping/enable
//     PlcTask Inputs/MAIN.force_rb_X[33] <-> Status process data mapping/force_rb_X
//     PlcTask Inputs/MAIN.force_rb_Y[33] <-> Status process data mapping/force_rb_Y
//     PlcTask Inputs/MAIN.force_rb_Z[33] <-> Status process data mapping/force_rb_Z
//     PlcTask Inputs/MAIN.force_sp_X[33] <-> Status process data mapping/force_sp_X
//     PlcTask Inputs/MAIN.force_sp_Y[33] <-> Status process data mapping/force_sp_Y
//     PlcTask Inputs/MAIN.force_sp_Z[33] <-> Status process data mapping/force_sp_Z
//     PlcTask Inputs/MAIN.pwm1[33] <-> Status process data mapping/pwm1
//     PlcTask Inputs/MAIN.pwm2[33] <-> Status process data mapping/pwm2
//     PlcTask Inputs/MAIN.pwm3[33] <-> Status process data mapping/pwm3
//     PlcTask Outputs/MAIN.enable_cmd[33] <-> Control process data mapping/enable
//     PlcTask Outputs/MAIN.force_cmd_X[33] <-> Control process data mapping/force_sp_X
//     PlcTask Outputs/MAIN.force_cmd_Y[33] <-> Control process data mapping/force_sp_Y
//     PlcTask Outputs/MAIN.force_cmd_Z[33] <-> Control process data mapping/force_sp_Z
//     PlcTask Outputs/MAIN.msthb[36] <-> Control process data mapping/msthb
//   SAsetGains/SAsetGains Instance <-> Device 1 (EtherCAT)/Box 33 (m1eph)/Box 37 (m1sa)
//     PlcTask Inputs/MAIN.cloop_stat[34] <-> Status process data mapping/close_loop
//     PlcTask Inputs/MAIN.enable_stat[34] <-> Status process data mapping/enable
//     PlcTask Inputs/MAIN.force_rb_X[34] <-> Status process data mapping/force_rb_X
//     PlcTask Inputs/MAIN.force_rb_Y[34] <-> Status process data mapping/force_rb_Y
//     PlcTask Inputs/MAIN.force_rb_Z[34] <-> Status process data mapping/force_rb_Z
//     PlcTask Inputs/MAIN.force_sp_X[34] <-> Status process data mapping/force_sp_X
//     PlcTask Inputs/MAIN.force_sp_Y[34] <-> Status process data mapping/force_sp_Y
//     PlcTask Inputs/MAIN.force_sp_Z[34] <-> Status process data mapping/force_sp_Z
//     PlcTask Inputs/MAIN.pwm1[34] <-> Status process data mapping/pwm1
//     PlcTask Inputs/MAIN.pwm2[34] <-> Status process data mapping/pwm2
//     PlcTask Inputs/MAIN.pwm3[34] <-> Status process data mapping/pwm3
//     PlcTask Outputs/MAIN.enable_cmd[34] <-> Control process data mapping/enable
//     PlcTask Outputs/MAIN.force_cmd_X[34] <-> Control process data mapping/force_sp_X
//     PlcTask Outputs/MAIN.force_cmd_Y[34] <-> Control process data mapping/force_sp_Y
//     PlcTask Outputs/MAIN.force_cmd_Z[34] <-> Control process data mapping/force_sp_Z
//     PlcTask Outputs/MAIN.msthb[37] <-> Control process data mapping/msthb
//   SAsetGains/SAsetGains Instance <-> Device 1 (EtherCAT)/Box 33 (m1eph)/Box 38 (m1sa)
//     PlcTask Inputs/MAIN.cloop_stat[35] <-> Status process data mapping/close_loop
//     PlcTask Inputs/MAIN.enable_stat[35] <-> Status process data mapping/enable
//     PlcTask Inputs/MAIN.force_rb_X[35] <-> Status process data mapping/force_rb_X
//     PlcTask Inputs/MAIN.force_rb_Y[35] <-> Status process data mapping/force_rb_Y
//     PlcTask Inputs/MAIN.force_rb_Z[35] <-> Status process data mapping/force_rb_Z
//     PlcTask Inputs/MAIN.force_sp_X[35] <-> Status process data mapping/force_sp_X
//     PlcTask Inputs/MAIN.force_sp_Y[35] <-> Status process data mapping/force_sp_Y
//     PlcTask Inputs/MAIN.force_sp_Z[35] <-> Status process data mapping/force_sp_Z
//     PlcTask Inputs/MAIN.pwm1[35] <-> Status process data mapping/pwm1
//     PlcTask Inputs/MAIN.pwm2[35] <-> Status process data mapping/pwm2
//     PlcTask Inputs/MAIN.pwm3[35] <-> Status process data mapping/pwm3
//     PlcTask Outputs/MAIN.enable_cmd[35] <-> Control process data mapping/enable
//     PlcTask Outputs/MAIN.force_cmd_X[35] <-> Control process data mapping/force_sp_X
//     PlcTask Outputs/MAIN.force_cmd_Y[35] <-> Control process data mapping/force_sp_Y
//     PlcTask Outputs/MAIN.force_cmd_Z[35] <-> Control process data mapping/force_sp_Z
//     PlcTask Outputs/MAIN.msthb[38] <-> Control process data mapping/msthb
//   SAsetGains/SAsetGains Instance <-> Device 1 (EtherCAT)/Box 33 (m1eph)/Box 39 (m1sa)
//     PlcTask Inputs/MAIN.cloop_stat[36] <-> Status process data mapping/close_loop
//     PlcTask Inputs/MAIN.enable_stat[36] <-> Status process data mapping/enable
//     PlcTask Inputs/MAIN.force_rb_X[36] <-> Status process data mapping/force_rb_X
//     PlcTask Inputs/MAIN.force_rb_Y[36] <-> Status process data mapping/force_rb_Y
//     PlcTask Inputs/MAIN.force_rb_Z[36] <-> Status process data mapping/force_rb_Z
//     PlcTask Inputs/MAIN.force_sp_X[36] <-> Status process data mapping/force_sp_X
//     PlcTask Inputs/MAIN.force_sp_Y[36] <-> Status process data mapping/force_sp_Y
//     PlcTask Inputs/MAIN.force_sp_Z[36] <-> Status process data mapping/force_sp_Z
//     PlcTask Inputs/MAIN.pwm1[36] <-> Status process data mapping/pwm1
//     PlcTask Inputs/MAIN.pwm2[36] <-> Status process data mapping/pwm2
//     PlcTask Inputs/MAIN.pwm3[36] <-> Status process data mapping/pwm3
//     PlcTask Outputs/MAIN.enable_cmd[36] <-> Control process data mapping/enable
//     PlcTask Outputs/MAIN.force_cmd_X[36] <-> Control process data mapping/force_sp_X
//     PlcTask Outputs/MAIN.force_cmd_Y[36] <-> Control process data mapping/force_sp_Y
//     PlcTask Outputs/MAIN.force_cmd_Z[36] <-> Control process data mapping/force_sp_Z
//     PlcTask Outputs/MAIN.msthb[39] <-> Control process data mapping/msthb
//   SAsetGains/SAsetGains Instance <-> Device 1 (EtherCAT)/Box 33 (m1eph)/Box 40 (m1sa)
//     PlcTask Inputs/MAIN.cloop_stat[37] <-> Status process data mapping/close_loop
//     PlcTask Inputs/MAIN.enable_stat[37] <-> Status process data mapping/enable
//     PlcTask Inputs/MAIN.force_rb_X[37] <-> Status process data mapping/force_rb_X
//     PlcTask Inputs/MAIN.force_rb_Y[37] <-> Status process data mapping/force_rb_Y
//     PlcTask Inputs/MAIN.force_rb_Z[37] <-> Status process data mapping/force_rb_Z
//     PlcTask Inputs/MAIN.force_sp_X[37] <-> Status process data mapping/force_sp_X
//     PlcTask Inputs/MAIN.force_sp_Y[37] <-> Status process data mapping/force_sp_Y
//     PlcTask Inputs/MAIN.force_sp_Z[37] <-> Status process data mapping/force_sp_Z
//     PlcTask Inputs/MAIN.pwm1[37] <-> Status process data mapping/pwm1
//     PlcTask Inputs/MAIN.pwm2[37] <-> Status process data mapping/pwm2
//     PlcTask Inputs/MAIN.pwm3[37] <-> Status process data mapping/pwm3
//     PlcTask Outputs/MAIN.enable_cmd[37] <-> Control process data mapping/enable
//     PlcTask Outputs/MAIN.force_cmd_X[37] <-> Control process data mapping/force_sp_X
//     PlcTask Outputs/MAIN.force_cmd_Y[37] <-> Control process data mapping/force_sp_Y
//     PlcTask Outputs/MAIN.force_cmd_Z[37] <-> Control process data mapping/force_sp_Z
//     PlcTask Outputs/MAIN.msthb[40] <-> Control process data mapping/msthb
//   SAsetGains/SAsetGains Instance <-> Device 1 (EtherCAT)/Box 33 (m1eph)/Box 41 (m1sa)
//     PlcTask Inputs/MAIN.cloop_stat[38] <-> Status process data mapping/close_loop
//     PlcTask Inputs/MAIN.enable_stat[38] <-> Status process data mapping/enable
//     PlcTask Inputs/MAIN.force_rb_X[38] <-> Status process data mapping/force_rb_X
//     PlcTask Inputs/MAIN.force_rb_Y[38] <-> Status process data mapping/force_rb_Y
//     PlcTask Inputs/MAIN.force_rb_Z[38] <-> Status process data mapping/force_rb_Z
//     PlcTask Inputs/MAIN.force_sp_X[38] <-> Status process data mapping/force_sp_X
//     PlcTask Inputs/MAIN.force_sp_Y[38] <-> Status process data mapping/force_sp_Y
//     PlcTask Inputs/MAIN.force_sp_Z[38] <-> Status process data mapping/force_sp_Z
//     PlcTask Inputs/MAIN.pwm1[38] <-> Status process data mapping/pwm1
//     PlcTask Inputs/MAIN.pwm2[38] <-> Status process data mapping/pwm2
//     PlcTask Inputs/MAIN.pwm3[38] <-> Status process data mapping/pwm3
//     PlcTask Outputs/MAIN.enable_cmd[38] <-> Control process data mapping/enable
//     PlcTask Outputs/MAIN.force_cmd_X[38] <-> Control process data mapping/force_sp_X
//     PlcTask Outputs/MAIN.force_cmd_Y[38] <-> Control process data mapping/force_sp_Y
//     PlcTask Outputs/MAIN.force_cmd_Z[38] <-> Control process data mapping/force_sp_Z
//     PlcTask Outputs/MAIN.msthb[41] <-> Control process data mapping/msthb
//   SAsetGains/SAsetGains Instance <-> Device 1 (EtherCAT)/Box 33 (m1eph)/Box 42 (m1sa)
//     PlcTask Inputs/MAIN.cloop_stat[39] <-> Status process data mapping/close_loop
//     PlcTask Inputs/MAIN.enable_stat[39] <-> Status process data mapping/enable
//     PlcTask Inputs/MAIN.force_rb_X[39] <-> Status process data mapping/force_rb_X
//     PlcTask Inputs/MAIN.force_rb_Y[39] <-> Status process data mapping/force_rb_Y
//     PlcTask Inputs/MAIN.force_rb_Z[39] <-> Status process data mapping/force_rb_Z
//     PlcTask Inputs/MAIN.force_sp_X[39] <-> Status process data mapping/force_sp_X
//     PlcTask Inputs/MAIN.force_sp_Y[39] <-> Status process data mapping/force_sp_Y
//     PlcTask Inputs/MAIN.force_sp_Z[39] <-> Status process data mapping/force_sp_Z
//     PlcTask Inputs/MAIN.pwm1[39] <-> Status process data mapping/pwm1
//     PlcTask Inputs/MAIN.pwm2[39] <-> Status process data mapping/pwm2
//     PlcTask Inputs/MAIN.pwm3[39] <-> Status process data mapping/pwm3
//     PlcTask Outputs/MAIN.enable_cmd[39] <-> Control process data mapping/enable
//     PlcTask Outputs/MAIN.force_cmd_X[39] <-> Control process data mapping/force_sp_X
//     PlcTask Outputs/MAIN.force_cmd_Y[39] <-> Control process data mapping/force_sp_Y
//     PlcTask Outputs/MAIN.force_cmd_Z[39] <-> Control process data mapping/force_sp_Z
//     PlcTask Outputs/MAIN.msthb[42] <-> Control process data mapping/msthb
//   SAsetGains/SAsetGains Instance <-> Device 1 (EtherCAT)/Box 33 (m1eph)/Box 43 (m1sa)
//     PlcTask Inputs/MAIN.cloop_stat[40] <-> Status process data mapping/close_loop
//     PlcTask Inputs/MAIN.enable_stat[40] <-> Status process data mapping/enable
//     PlcTask Inputs/MAIN.force_rb_X[40] <-> Status process data mapping/force_rb_X
//     PlcTask Inputs/MAIN.force_rb_Y[40] <-> Status process data mapping/force_rb_Y
//     PlcTask Inputs/MAIN.force_rb_Z[40] <-> Status process data mapping/force_rb_Z
//     PlcTask Inputs/MAIN.force_sp_X[40] <-> Status process data mapping/force_sp_X
//     PlcTask Inputs/MAIN.force_sp_Y[40] <-> Status process data mapping/force_sp_Y
//     PlcTask Inputs/MAIN.force_sp_Z[40] <-> Status process data mapping/force_sp_Z
//     PlcTask Inputs/MAIN.pwm1[40] <-> Status process data mapping/pwm1
//     PlcTask Inputs/MAIN.pwm2[40] <-> Status process data mapping/pwm2
//     PlcTask Inputs/MAIN.pwm3[40] <-> Status process data mapping/pwm3
//     PlcTask Outputs/MAIN.enable_cmd[40] <-> Control process data mapping/enable
//     PlcTask Outputs/MAIN.force_cmd_X[40] <-> Control process data mapping/force_sp_X
//     PlcTask Outputs/MAIN.force_cmd_Y[40] <-> Control process data mapping/force_sp_Y
//     PlcTask Outputs/MAIN.force_cmd_Z[40] <-> Control process data mapping/force_sp_Z
//     PlcTask Outputs/MAIN.msthb[43] <-> Control process data mapping/msthb
//   SAsetGains/SAsetGains Instance <-> Device 1 (EtherCAT)/Box 33 (m1eph)/Box 44 (m1sa)
//     PlcTask Inputs/MAIN.cloop_stat[41] <-> Status process data mapping/close_loop
//     PlcTask Inputs/MAIN.enable_stat[41] <-> Status process data mapping/enable
//     PlcTask Inputs/MAIN.force_rb_X[41] <-> Status process data mapping/force_rb_X
//     PlcTask Inputs/MAIN.force_rb_Y[41] <-> Status process data mapping/force_rb_Y
//     PlcTask Inputs/MAIN.force_rb_Z[41] <-> Status process data mapping/force_rb_Z
//     PlcTask Inputs/MAIN.force_sp_X[41] <-> Status process data mapping/force_sp_X
//     PlcTask Inputs/MAIN.force_sp_Y[41] <-> Status process data mapping/force_sp_Y
//     PlcTask Inputs/MAIN.force_sp_Z[41] <-> Status process data mapping/force_sp_Z
//     PlcTask Inputs/MAIN.pwm1[41] <-> Status process data mapping/pwm1
//     PlcTask Inputs/MAIN.pwm2[41] <-> Status process data mapping/pwm2
//     PlcTask Inputs/MAIN.pwm3[41] <-> Status process data mapping/pwm3
//     PlcTask Outputs/MAIN.enable_cmd[41] <-> Control process data mapping/enable
//     PlcTask Outputs/MAIN.force_cmd_X[41] <-> Control process data mapping/force_sp_X
//     PlcTask Outputs/MAIN.force_cmd_Y[41] <-> Control process data mapping/force_sp_Y
//     PlcTask Outputs/MAIN.force_cmd_Z[41] <-> Control process data mapping/force_sp_Z
//     PlcTask Outputs/MAIN.msthb[44] <-> Control process data mapping/msthb
//   SAsetGains/SAsetGains Instance <-> Device 1 (EtherCAT)/Box 33 (m1eph)/Box 45 (m1sa)
//     PlcTask Inputs/MAIN.cloop_stat[42] <-> Status process data mapping/close_loop
//     PlcTask Inputs/MAIN.enable_stat[42] <-> Status process data mapping/enable
//     PlcTask Inputs/MAIN.force_rb_X[42] <-> Status process data mapping/force_rb_X
//     PlcTask Inputs/MAIN.force_rb_Y[42] <-> Status process data mapping/force_rb_Y
//     PlcTask Inputs/MAIN.force_rb_Z[42] <-> Status process data mapping/force_rb_Z
//     PlcTask Inputs/MAIN.force_sp_X[42] <-> Status process data mapping/force_sp_X
//     PlcTask Inputs/MAIN.force_sp_Y[42] <-> Status process data mapping/force_sp_Y
//     PlcTask Inputs/MAIN.force_sp_Z[42] <-> Status process data mapping/force_sp_Z
//     PlcTask Inputs/MAIN.pwm1[42] <-> Status process data mapping/pwm1
//     PlcTask Inputs/MAIN.pwm2[42] <-> Status process data mapping/pwm2
//     PlcTask Inputs/MAIN.pwm3[42] <-> Status process data mapping/pwm3
//     PlcTask Outputs/MAIN.enable_cmd[42] <-> Control process data mapping/enable
//     PlcTask Outputs/MAIN.force_cmd_X[42] <-> Control process data mapping/force_sp_X
//     PlcTask Outputs/MAIN.force_cmd_Y[42] <-> Control process data mapping/force_sp_Y
//     PlcTask Outputs/MAIN.force_cmd_Z[42] <-> Control process data mapping/force_sp_Z
//     PlcTask Outputs/MAIN.msthb[45] <-> Control process data mapping/msthb
//   SAsetGains/SAsetGains Instance <-> Device 1 (EtherCAT)/Box 46 (m1eph)
//     PlcTask Outputs/MAIN.msthb[46] <-> Control process data mapping/msthb
//   SAsetGains/SAsetGains Instance <-> Device 1 (EtherCAT)/Box 46 (m1eph)/Box 47 (m1sa)
//     PlcTask Inputs/MAIN.cloop_stat[43] <-> Status process data mapping/close_loop
//     PlcTask Inputs/MAIN.enable_stat[43] <-> Status process data mapping/enable
//     PlcTask Inputs/MAIN.force_rb_X[43] <-> Status process data mapping/force_rb_X
//     PlcTask Inputs/MAIN.force_rb_Y[43] <-> Status process data mapping/force_rb_Y
//     PlcTask Inputs/MAIN.force_rb_Z[43] <-> Status process data mapping/force_rb_Z
//     PlcTask Inputs/MAIN.force_sp_X[43] <-> Status process data mapping/force_sp_X
//     PlcTask Inputs/MAIN.force_sp_Y[43] <-> Status process data mapping/force_sp_Y
//     PlcTask Inputs/MAIN.force_sp_Z[43] <-> Status process data mapping/force_sp_Z
//     PlcTask Inputs/MAIN.pwm1[43] <-> Status process data mapping/pwm1
//     PlcTask Inputs/MAIN.pwm2[43] <-> Status process data mapping/pwm2
//     PlcTask Inputs/MAIN.pwm3[43] <-> Status process data mapping/pwm3
//     PlcTask Outputs/MAIN.enable_cmd[43] <-> Control process data mapping/enable
//     PlcTask Outputs/MAIN.force_cmd_X[43] <-> Control process data mapping/force_sp_X
//     PlcTask Outputs/MAIN.force_cmd_Y[43] <-> Control process data mapping/force_sp_Y
//     PlcTask Outputs/MAIN.force_cmd_Z[43] <-> Control process data mapping/force_sp_Z
//     PlcTask Outputs/MAIN.msthb[47] <-> Control process data mapping/msthb
//   SAsetGains/SAsetGains Instance <-> Device 1 (EtherCAT)/Box 46 (m1eph)/Box 48 (m1sa)
//     PlcTask Inputs/MAIN.cloop_stat[44] <-> Status process data mapping/close_loop
//     PlcTask Inputs/MAIN.enable_stat[44] <-> Status process data mapping/enable
//     PlcTask Inputs/MAIN.force_rb_X[44] <-> Status process data mapping/force_rb_X
//     PlcTask Inputs/MAIN.force_rb_Y[44] <-> Status process data mapping/force_rb_Y
//     PlcTask Inputs/MAIN.force_rb_Z[44] <-> Status process data mapping/force_rb_Z
//     PlcTask Inputs/MAIN.force_sp_X[44] <-> Status process data mapping/force_sp_X
//     PlcTask Inputs/MAIN.force_sp_Y[44] <-> Status process data mapping/force_sp_Y
//     PlcTask Inputs/MAIN.force_sp_Z[44] <-> Status process data mapping/force_sp_Z
//     PlcTask Inputs/MAIN.pwm1[44] <-> Status process data mapping/pwm1
//     PlcTask Inputs/MAIN.pwm2[44] <-> Status process data mapping/pwm2
//     PlcTask Inputs/MAIN.pwm3[44] <-> Status process data mapping/pwm3
//     PlcTask Outputs/MAIN.enable_cmd[44] <-> Control process data mapping/enable
//     PlcTask Outputs/MAIN.force_cmd_X[44] <-> Control process data mapping/force_sp_X
//     PlcTask Outputs/MAIN.force_cmd_Y[44] <-> Control process data mapping/force_sp_Y
//     PlcTask Outputs/MAIN.force_cmd_Z[44] <-> Control process data mapping/force_sp_Z
//     PlcTask Outputs/MAIN.msthb[48] <-> Control process data mapping/msthb
//   SAsetGains/SAsetGains Instance <-> Device 1 (EtherCAT)/Box 46 (m1eph)/Box 49 (m1sa)
//     PlcTask Inputs/MAIN.cloop_stat[45] <-> Status process data mapping/close_loop
//     PlcTask Inputs/MAIN.enable_stat[45] <-> Status process data mapping/enable
//     PlcTask Inputs/MAIN.force_rb_X[45] <-> Status process data mapping/force_rb_X
//     PlcTask Inputs/MAIN.force_rb_Y[45] <-> Status process data mapping/force_rb_Y
//     PlcTask Inputs/MAIN.force_rb_Z[45] <-> Status process data mapping/force_rb_Z
//     PlcTask Inputs/MAIN.force_sp_X[45] <-> Status process data mapping/force_sp_X
//     PlcTask Inputs/MAIN.force_sp_Y[45] <-> Status process data mapping/force_sp_Y
//     PlcTask Inputs/MAIN.force_sp_Z[45] <-> Status process data mapping/force_sp_Z
//     PlcTask Inputs/MAIN.pwm1[45] <-> Status process data mapping/pwm1
//     PlcTask Inputs/MAIN.pwm2[45] <-> Status process data mapping/pwm2
//     PlcTask Inputs/MAIN.pwm3[45] <-> Status process data mapping/pwm3
//     PlcTask Outputs/MAIN.enable_cmd[45] <-> Control process data mapping/enable
//     PlcTask Outputs/MAIN.force_cmd_X[45] <-> Control process data mapping/force_sp_X
//     PlcTask Outputs/MAIN.force_cmd_Y[45] <-> Control process data mapping/force_sp_Y
//     PlcTask Outputs/MAIN.force_cmd_Z[45] <-> Control process data mapping/force_sp_Z
//     PlcTask Outputs/MAIN.msthb[49] <-> Control process data mapping/msthb
//   SAsetGains/SAsetGains Instance <-> Device 1 (EtherCAT)/Box 46 (m1eph)/Box 50 (m1sa)
//     PlcTask Inputs/MAIN.cloop_stat[46] <-> Status process data mapping/close_loop
//     PlcTask Inputs/MAIN.enable_stat[46] <-> Status process data mapping/enable
//     PlcTask Inputs/MAIN.force_rb_X[46] <-> Status process data mapping/force_rb_X
//     PlcTask Inputs/MAIN.force_rb_Y[46] <-> Status process data mapping/force_rb_Y
//     PlcTask Inputs/MAIN.force_rb_Z[46] <-> Status process data mapping/force_rb_Z
//     PlcTask Inputs/MAIN.force_sp_X[46] <-> Status process data mapping/force_sp_X
//     PlcTask Inputs/MAIN.force_sp_Y[46] <-> Status process data mapping/force_sp_Y
//     PlcTask Inputs/MAIN.force_sp_Z[46] <-> Status process data mapping/force_sp_Z
//     PlcTask Inputs/MAIN.pwm1[46] <-> Status process data mapping/pwm1
//     PlcTask Inputs/MAIN.pwm2[46] <-> Status process data mapping/pwm2
//     PlcTask Inputs/MAIN.pwm3[46] <-> Status process data mapping/pwm3
//     PlcTask Outputs/MAIN.enable_cmd[46] <-> Control process data mapping/enable
//     PlcTask Outputs/MAIN.force_cmd_X[46] <-> Control process data mapping/force_sp_X
//     PlcTask Outputs/MAIN.force_cmd_Y[46] <-> Control process data mapping/force_sp_Y
//     PlcTask Outputs/MAIN.force_cmd_Z[46] <-> Control process data mapping/force_sp_Z
//     PlcTask Outputs/MAIN.msthb[50] <-> Control process data mapping/msthb
//   SAsetGains/SAsetGains Instance <-> Device 1 (EtherCAT)/Box 46 (m1eph)/Box 51 (m1sa)
//     PlcTask Inputs/MAIN.cloop_stat[47] <-> Status process data mapping/close_loop
//     PlcTask Inputs/MAIN.enable_stat[47] <-> Status process data mapping/enable
//     PlcTask Inputs/MAIN.force_rb_X[47] <-> Status process data mapping/force_rb_X
//     PlcTask Inputs/MAIN.force_rb_Y[47] <-> Status process data mapping/force_rb_Y
//     PlcTask Inputs/MAIN.force_rb_Z[47] <-> Status process data mapping/force_rb_Z
//     PlcTask Inputs/MAIN.force_sp_X[47] <-> Status process data mapping/force_sp_X
//     PlcTask Inputs/MAIN.force_sp_Y[47] <-> Status process data mapping/force_sp_Y
//     PlcTask Inputs/MAIN.force_sp_Z[47] <-> Status process data mapping/force_sp_Z
//     PlcTask Inputs/MAIN.pwm1[47] <-> Status process data mapping/pwm1
//     PlcTask Inputs/MAIN.pwm2[47] <-> Status process data mapping/pwm2
//     PlcTask Inputs/MAIN.pwm3[47] <-> Status process data mapping/pwm3
//     PlcTask Outputs/MAIN.enable_cmd[47] <-> Control process data mapping/enable
//     PlcTask Outputs/MAIN.force_cmd_X[47] <-> Control process data mapping/force_sp_X
//     PlcTask Outputs/MAIN.force_cmd_Y[47] <-> Control process data mapping/force_sp_Y
//     PlcTask Outputs/MAIN.force_cmd_Z[47] <-> Control process data mapping/force_sp_Z
//     PlcTask Outputs/MAIN.msthb[51] <-> Control process data mapping/msthb
//   SAsetGains/SAsetGains Instance <-> Device 1 (EtherCAT)/Box 46 (m1eph)/Box 52 (m1sa)
//     PlcTask Inputs/MAIN.cloop_stat[48] <-> Status process data mapping/close_loop
//     PlcTask Inputs/MAIN.enable_stat[48] <-> Status process data mapping/enable
//     PlcTask Inputs/MAIN.force_rb_X[48] <-> Status process data mapping/force_rb_X
//     PlcTask Inputs/MAIN.force_rb_Y[48] <-> Status process data mapping/force_rb_Y
//     PlcTask Inputs/MAIN.force_rb_Z[48] <-> Status process data mapping/force_rb_Z
//     PlcTask Inputs/MAIN.force_sp_X[48] <-> Status process data mapping/force_sp_X
//     PlcTask Inputs/MAIN.force_sp_Y[48] <-> Status process data mapping/force_sp_Y
//     PlcTask Inputs/MAIN.force_sp_Z[48] <-> Status process data mapping/force_sp_Z
//     PlcTask Inputs/MAIN.pwm1[48] <-> Status process data mapping/pwm1
//     PlcTask Inputs/MAIN.pwm2[48] <-> Status process data mapping/pwm2
//     PlcTask Inputs/MAIN.pwm3[48] <-> Status process data mapping/pwm3
//     PlcTask Outputs/MAIN.enable_cmd[48] <-> Control process data mapping/enable
//     PlcTask Outputs/MAIN.force_cmd_X[48] <-> Control process data mapping/force_sp_X
//     PlcTask Outputs/MAIN.force_cmd_Y[48] <-> Control process data mapping/force_sp_Y
//     PlcTask Outputs/MAIN.force_cmd_Z[48] <-> Control process data mapping/force_sp_Z
//     PlcTask Outputs/MAIN.msthb[52] <-> Control process data mapping/msthb
//   SAsetGains/SAsetGains Instance <-> Device 1 (EtherCAT)/Box 46 (m1eph)/Box 53 (m1sa)
//     PlcTask Inputs/MAIN.cloop_stat[49] <-> Status process data mapping/close_loop
//     PlcTask Inputs/MAIN.enable_stat[49] <-> Status process data mapping/enable
//     PlcTask Inputs/MAIN.force_rb_X[49] <-> Status process data mapping/force_rb_X
//     PlcTask Inputs/MAIN.force_rb_Y[49] <-> Status process data mapping/force_rb_Y
//     PlcTask Inputs/MAIN.force_rb_Z[49] <-> Status process data mapping/force_rb_Z
//     PlcTask Inputs/MAIN.force_sp_X[49] <-> Status process data mapping/force_sp_X
//     PlcTask Inputs/MAIN.force_sp_Y[49] <-> Status process data mapping/force_sp_Y
//     PlcTask Inputs/MAIN.force_sp_Z[49] <-> Status process data mapping/force_sp_Z
//     PlcTask Inputs/MAIN.pwm1[49] <-> Status process data mapping/pwm1
//     PlcTask Inputs/MAIN.pwm2[49] <-> Status process data mapping/pwm2
//     PlcTask Inputs/MAIN.pwm3[49] <-> Status process data mapping/pwm3
//     PlcTask Outputs/MAIN.enable_cmd[49] <-> Control process data mapping/enable
//     PlcTask Outputs/MAIN.force_cmd_X[49] <-> Control process data mapping/force_sp_X
//     PlcTask Outputs/MAIN.force_cmd_Y[49] <-> Control process data mapping/force_sp_Y
//     PlcTask Outputs/MAIN.force_cmd_Z[49] <-> Control process data mapping/force_sp_Z
//     PlcTask Outputs/MAIN.msthb[53] <-> Control process data mapping/msthb
//   SAsetGains/SAsetGains Instance <-> Device 1 (EtherCAT)/Box 46 (m1eph)/Box 54 (m1sa)
//     PlcTask Inputs/MAIN.cloop_stat[50] <-> Status process data mapping/close_loop
//     PlcTask Inputs/MAIN.enable_stat[50] <-> Status process data mapping/enable
//     PlcTask Inputs/MAIN.force_rb_X[50] <-> Status process data mapping/force_rb_X
//     PlcTask Inputs/MAIN.force_rb_Y[50] <-> Status process data mapping/force_rb_Y
//     PlcTask Inputs/MAIN.force_rb_Z[50] <-> Status process data mapping/force_rb_Z
//     PlcTask Inputs/MAIN.force_sp_X[50] <-> Status process data mapping/force_sp_X
//     PlcTask Inputs/MAIN.force_sp_Y[50] <-> Status process data mapping/force_sp_Y
//     PlcTask Inputs/MAIN.force_sp_Z[50] <-> Status process data mapping/force_sp_Z
//     PlcTask Inputs/MAIN.pwm1[50] <-> Status process data mapping/pwm1
//     PlcTask Inputs/MAIN.pwm2[50] <-> Status process data mapping/pwm2
//     PlcTask Inputs/MAIN.pwm3[50] <-> Status process data mapping/pwm3
//     PlcTask Outputs/MAIN.enable_cmd[50] <-> Control process data mapping/enable
//     PlcTask Outputs/MAIN.force_cmd_X[50] <-> Control process data mapping/force_sp_X
//     PlcTask Outputs/MAIN.force_cmd_Y[50] <-> Control process data mapping/force_sp_Y
//     PlcTask Outputs/MAIN.force_cmd_Z[50] <-> Control process data mapping/force_sp_Z
//     PlcTask Outputs/MAIN.msthb[54] <-> Control process data mapping/msthb
//   SAsetGains/SAsetGains Instance <-> Device 1 (EtherCAT)/Box 46 (m1eph)/Box 55 (m1sa)
//     PlcTask Inputs/MAIN.cloop_stat[51] <-> Status process data mapping/close_loop
//     PlcTask Inputs/MAIN.enable_stat[51] <-> Status process data mapping/enable
//     PlcTask Inputs/MAIN.force_rb_X[51] <-> Status process data mapping/force_rb_X
//     PlcTask Inputs/MAIN.force_rb_Y[51] <-> Status process data mapping/force_rb_Y
//     PlcTask Inputs/MAIN.force_rb_Z[51] <-> Status process data mapping/force_rb_Z
//     PlcTask Inputs/MAIN.force_sp_X[51] <-> Status process data mapping/force_sp_X
//     PlcTask Inputs/MAIN.force_sp_Y[51] <-> Status process data mapping/force_sp_Y
//     PlcTask Inputs/MAIN.force_sp_Z[51] <-> Status process data mapping/force_sp_Z
//     PlcTask Inputs/MAIN.pwm1[51] <-> Status process data mapping/pwm1
//     PlcTask Inputs/MAIN.pwm2[51] <-> Status process data mapping/pwm2
//     PlcTask Inputs/MAIN.pwm3[51] <-> Status process data mapping/pwm3
//     PlcTask Outputs/MAIN.enable_cmd[51] <-> Control process data mapping/enable
//     PlcTask Outputs/MAIN.force_cmd_X[51] <-> Control process data mapping/force_sp_X
//     PlcTask Outputs/MAIN.force_cmd_Y[51] <-> Control process data mapping/force_sp_Y
//     PlcTask Outputs/MAIN.force_cmd_Z[51] <-> Control process data mapping/force_sp_Z
//     PlcTask Outputs/MAIN.msthb[55] <-> Control process data mapping/msthb
//   SAsetGains/SAsetGains Instance <-> Device 1 (EtherCAT)/Box 46 (m1eph)/Box 56 (m1sa)
//     PlcTask Inputs/MAIN.cloop_stat[52] <-> Status process data mapping/close_loop
//     PlcTask Inputs/MAIN.enable_stat[52] <-> Status process data mapping/enable
//     PlcTask Inputs/MAIN.force_rb_X[52] <-> Status process data mapping/force_rb_X
//     PlcTask Inputs/MAIN.force_rb_Y[52] <-> Status process data mapping/force_rb_Y
//     PlcTask Inputs/MAIN.force_rb_Z[52] <-> Status process data mapping/force_rb_Z
//     PlcTask Inputs/MAIN.force_sp_X[52] <-> Status process data mapping/force_sp_X
//     PlcTask Inputs/MAIN.force_sp_Y[52] <-> Status process data mapping/force_sp_Y
//     PlcTask Inputs/MAIN.force_sp_Z[52] <-> Status process data mapping/force_sp_Z
//     PlcTask Inputs/MAIN.pwm1[52] <-> Status process data mapping/pwm1
//     PlcTask Inputs/MAIN.pwm2[52] <-> Status process data mapping/pwm2
//     PlcTask Inputs/MAIN.pwm3[52] <-> Status process data mapping/pwm3
//     PlcTask Outputs/MAIN.enable_cmd[52] <-> Control process data mapping/enable
//     PlcTask Outputs/MAIN.force_cmd_X[52] <-> Control process data mapping/force_sp_X
//     PlcTask Outputs/MAIN.force_cmd_Y[52] <-> Control process data mapping/force_sp_Y
//     PlcTask Outputs/MAIN.force_cmd_Z[52] <-> Control process data mapping/force_sp_Z
//     PlcTask Outputs/MAIN.msthb[56] <-> Control process data mapping/msthb
//   SAsetGains/SAsetGains Instance <-> Device 1 (EtherCAT)/Box 46 (m1eph)/Box 57 (m1sa)
//     PlcTask Inputs/MAIN.cloop_stat[53] <-> Status process data mapping/close_loop
//     PlcTask Inputs/MAIN.enable_stat[53] <-> Status process data mapping/enable
//     PlcTask Inputs/MAIN.force_rb_X[53] <-> Status process data mapping/force_rb_X
//     PlcTask Inputs/MAIN.force_rb_Y[53] <-> Status process data mapping/force_rb_Y
//     PlcTask Inputs/MAIN.force_rb_Z[53] <-> Status process data mapping/force_rb_Z
//     PlcTask Inputs/MAIN.force_sp_X[53] <-> Status process data mapping/force_sp_X
//     PlcTask Inputs/MAIN.force_sp_Y[53] <-> Status process data mapping/force_sp_Y
//     PlcTask Inputs/MAIN.force_sp_Z[53] <-> Status process data mapping/force_sp_Z
//     PlcTask Inputs/MAIN.pwm1[53] <-> Status process data mapping/pwm1
//     PlcTask Inputs/MAIN.pwm2[53] <-> Status process data mapping/pwm2
//     PlcTask Inputs/MAIN.pwm3[53] <-> Status process data mapping/pwm3
//     PlcTask Outputs/MAIN.enable_cmd[53] <-> Control process data mapping/enable
//     PlcTask Outputs/MAIN.force_cmd_X[53] <-> Control process data mapping/force_sp_X
//     PlcTask Outputs/MAIN.force_cmd_Y[53] <-> Control process data mapping/force_sp_Y
//     PlcTask Outputs/MAIN.force_cmd_Z[53] <-> Control process data mapping/force_sp_Z
//     PlcTask Outputs/MAIN.msthb[57] <-> Control process data mapping/msthb
//   SAsetGains/SAsetGains Instance <-> Device 1 (EtherCAT)/Box 46 (m1eph)/Box 58 (m1sa)
//     PlcTask Inputs/MAIN.cloop_stat[54] <-> Status process data mapping/close_loop
//     PlcTask Inputs/MAIN.enable_stat[54] <-> Status process data mapping/enable
//     PlcTask Inputs/MAIN.force_rb_X[54] <-> Status process data mapping/force_rb_X
//     PlcTask Inputs/MAIN.force_rb_Y[54] <-> Status process data mapping/force_rb_Y
//     PlcTask Inputs/MAIN.force_rb_Z[54] <-> Status process data mapping/force_rb_Z
//     PlcTask Inputs/MAIN.force_sp_X[54] <-> Status process data mapping/force_sp_X
//     PlcTask Inputs/MAIN.force_sp_Y[54] <-> Status process data mapping/force_sp_Y
//     PlcTask Inputs/MAIN.force_sp_Z[54] <-> Status process data mapping/force_sp_Z
//     PlcTask Inputs/MAIN.pwm1[54] <-> Status process data mapping/pwm1
//     PlcTask Inputs/MAIN.pwm2[54] <-> Status process data mapping/pwm2
//     PlcTask Inputs/MAIN.pwm3[54] <-> Status process data mapping/pwm3
//     PlcTask Outputs/MAIN.enable_cmd[54] <-> Control process data mapping/enable
//     PlcTask Outputs/MAIN.force_cmd_X[54] <-> Control process data mapping/force_sp_X
//     PlcTask Outputs/MAIN.force_cmd_Y[54] <-> Control process data mapping/force_sp_Y
//     PlcTask Outputs/MAIN.force_cmd_Z[54] <-> Control process data mapping/force_sp_Z
//     PlcTask Outputs/MAIN.msthb[58] <-> Control process data mapping/msthb
//   SAsetGains/SAsetGains Instance <-> Device 1 (EtherCAT)/Box 46 (m1eph)/Box 59 (m1sa)
//     PlcTask Inputs/MAIN.cloop_stat[55] <-> Status process data mapping/close_loop
//     PlcTask Inputs/MAIN.enable_stat[55] <-> Status process data mapping/enable
//     PlcTask Inputs/MAIN.force_rb_X[55] <-> Status process data mapping/force_rb_X
//     PlcTask Inputs/MAIN.force_rb_Y[55] <-> Status process data mapping/force_rb_Y
//     PlcTask Inputs/MAIN.force_rb_Z[55] <-> Status process data mapping/force_rb_Z
//     PlcTask Inputs/MAIN.force_sp_X[55] <-> Status process data mapping/force_sp_X
//     PlcTask Inputs/MAIN.force_sp_Y[55] <-> Status process data mapping/force_sp_Y
//     PlcTask Inputs/MAIN.force_sp_Z[55] <-> Status process data mapping/force_sp_Z
//     PlcTask Inputs/MAIN.pwm1[55] <-> Status process data mapping/pwm1
//     PlcTask Inputs/MAIN.pwm2[55] <-> Status process data mapping/pwm2
//     PlcTask Inputs/MAIN.pwm3[55] <-> Status process data mapping/pwm3
//     PlcTask Outputs/MAIN.enable_cmd[55] <-> Control process data mapping/enable
//     PlcTask Outputs/MAIN.force_cmd_X[55] <-> Control process data mapping/force_sp_X
//     PlcTask Outputs/MAIN.force_cmd_Y[55] <-> Control process data mapping/force_sp_Y
//     PlcTask Outputs/MAIN.force_cmd_Z[55] <-> Control process data mapping/force_sp_Z
//     PlcTask Outputs/MAIN.msthb[59] <-> Control process data mapping/msthb
//   SAsetGains/SAsetGains Instance <-> Device 1 (EtherCAT)/Box 46 (m1eph)/Box 60 (m1sa)
//     PlcTask Inputs/MAIN.cloop_stat[56] <-> Status process data mapping/close_loop
//     PlcTask Inputs/MAIN.enable_stat[56] <-> Status process data mapping/enable
//     PlcTask Inputs/MAIN.force_rb_X[56] <-> Status process data mapping/force_rb_X
//     PlcTask Inputs/MAIN.force_rb_Y[56] <-> Status process data mapping/force_rb_Y
//     PlcTask Inputs/MAIN.force_rb_Z[56] <-> Status process data mapping/force_rb_Z
//     PlcTask Inputs/MAIN.force_sp_X[56] <-> Status process data mapping/force_sp_X
//     PlcTask Inputs/MAIN.force_sp_Y[56] <-> Status process data mapping/force_sp_Y
//     PlcTask Inputs/MAIN.force_sp_Z[56] <-> Status process data mapping/force_sp_Z
//     PlcTask Inputs/MAIN.pwm1[56] <-> Status process data mapping/pwm1
//     PlcTask Inputs/MAIN.pwm2[56] <-> Status process data mapping/pwm2
//     PlcTask Inputs/MAIN.pwm3[56] <-> Status process data mapping/pwm3
//     PlcTask Outputs/MAIN.enable_cmd[56] <-> Control process data mapping/enable
//     PlcTask Outputs/MAIN.force_cmd_X[56] <-> Control process data mapping/force_sp_X
//     PlcTask Outputs/MAIN.force_cmd_Y[56] <-> Control process data mapping/force_sp_Y
//     PlcTask Outputs/MAIN.force_cmd_Z[56] <-> Control process data mapping/force_sp_Z
//     PlcTask Outputs/MAIN.msthb[60] <-> Control process data mapping/msthb
//   SAsetGains/SAsetGains Instance <-> Device 1 (EtherCAT)/Box 46 (m1eph)/Box 61 (m1sa)
//     PlcTask Inputs/MAIN.cloop_stat[57] <-> Status process data mapping/close_loop
//     PlcTask Inputs/MAIN.enable_stat[57] <-> Status process data mapping/enable
//     PlcTask Inputs/MAIN.force_rb_X[57] <-> Status process data mapping/force_rb_X
//     PlcTask Inputs/MAIN.force_rb_Y[57] <-> Status process data mapping/force_rb_Y
//     PlcTask Inputs/MAIN.force_rb_Z[57] <-> Status process data mapping/force_rb_Z
//     PlcTask Inputs/MAIN.force_sp_X[57] <-> Status process data mapping/force_sp_X
//     PlcTask Inputs/MAIN.force_sp_Y[57] <-> Status process data mapping/force_sp_Y
//     PlcTask Inputs/MAIN.force_sp_Z[57] <-> Status process data mapping/force_sp_Z
//     PlcTask Inputs/MAIN.pwm1[57] <-> Status process data mapping/pwm1
//     PlcTask Inputs/MAIN.pwm2[57] <-> Status process data mapping/pwm2
//     PlcTask Inputs/MAIN.pwm3[57] <-> Status process data mapping/pwm3
//     PlcTask Outputs/MAIN.enable_cmd[57] <-> Control process data mapping/enable
//     PlcTask Outputs/MAIN.force_cmd_X[57] <-> Control process data mapping/force_sp_X
//     PlcTask Outputs/MAIN.force_cmd_Y[57] <-> Control process data mapping/force_sp_Y
//     PlcTask Outputs/MAIN.force_cmd_Z[57] <-> Control process data mapping/force_sp_Z
//     PlcTask Outputs/MAIN.msthb[61] <-> Control process data mapping/msthb
//   SAsetGains/SAsetGains Instance <-> Device 1 (EtherCAT)/Box 46 (m1eph)/Box 62 (m1sa)
//     PlcTask Inputs/MAIN.cloop_stat[58] <-> Status process data mapping/close_loop
//     PlcTask Inputs/MAIN.enable_stat[58] <-> Status process data mapping/enable
//     PlcTask Inputs/MAIN.force_rb_X[58] <-> Status process data mapping/force_rb_X
//     PlcTask Inputs/MAIN.force_rb_Y[58] <-> Status process data mapping/force_rb_Y
//     PlcTask Inputs/MAIN.force_rb_Z[58] <-> Status process data mapping/force_rb_Z
//     PlcTask Inputs/MAIN.force_sp_X[58] <-> Status process data mapping/force_sp_X
//     PlcTask Inputs/MAIN.force_sp_Y[58] <-> Status process data mapping/force_sp_Y
//     PlcTask Inputs/MAIN.force_sp_Z[58] <-> Status process data mapping/force_sp_Z
//     PlcTask Inputs/MAIN.pwm1[58] <-> Status process data mapping/pwm1
//     PlcTask Inputs/MAIN.pwm2[58] <-> Status process data mapping/pwm2
//     PlcTask Inputs/MAIN.pwm3[58] <-> Status process data mapping/pwm3
//     PlcTask Outputs/MAIN.enable_cmd[58] <-> Control process data mapping/enable
//     PlcTask Outputs/MAIN.force_cmd_X[58] <-> Control process data mapping/force_sp_X
//     PlcTask Outputs/MAIN.force_cmd_Y[58] <-> Control process data mapping/force_sp_Y
//     PlcTask Outputs/MAIN.force_cmd_Z[58] <-> Control process data mapping/force_sp_Z
//     PlcTask Outputs/MAIN.msthb[62] <-> Control process data mapping/msthb
//   SAsetGains/SAsetGains Instance <-> Device 1 (EtherCAT)/Box 63 (m1eph)
//     PlcTask Outputs/MAIN.msthb[63] <-> Control process data mapping/msthb
//   SAsetGains/SAsetGains Instance <-> Device 1 (EtherCAT)/Box 63 (m1eph)/Box 64 (m1sa)
//     PlcTask Inputs/MAIN.cloop_stat[59] <-> Status process data mapping/close_loop
//     PlcTask Inputs/MAIN.enable_stat[59] <-> Status process data mapping/enable
//     PlcTask Inputs/MAIN.force_rb_X[59] <-> Status process data mapping/force_rb_X
//     PlcTask Inputs/MAIN.force_rb_Y[59] <-> Status process data mapping/force_rb_Y
//     PlcTask Inputs/MAIN.force_rb_Z[59] <-> Status process data mapping/force_rb_Z
//     PlcTask Inputs/MAIN.force_sp_X[59] <-> Status process data mapping/force_sp_X
//     PlcTask Inputs/MAIN.force_sp_Y[59] <-> Status process data mapping/force_sp_Y
//     PlcTask Inputs/MAIN.force_sp_Z[59] <-> Status process data mapping/force_sp_Z
//     PlcTask Inputs/MAIN.pwm1[59] <-> Status process data mapping/pwm1
//     PlcTask Inputs/MAIN.pwm2[59] <-> Status process data mapping/pwm2
//     PlcTask Inputs/MAIN.pwm3[59] <-> Status process data mapping/pwm3
//     PlcTask Outputs/MAIN.enable_cmd[59] <-> Control process data mapping/enable
//     PlcTask Outputs/MAIN.force_cmd_X[59] <-> Control process data mapping/force_sp_X
//     PlcTask Outputs/MAIN.force_cmd_Y[59] <-> Control process data mapping/force_sp_Y
//     PlcTask Outputs/MAIN.force_cmd_Z[59] <-> Control process data mapping/force_sp_Z
//     PlcTask Outputs/MAIN.msthb[64] <-> Control process data mapping/msthb
//   SAsetGains/SAsetGains Instance <-> Device 1 (EtherCAT)/Box 63 (m1eph)/Box 65 (m1sa)
//     PlcTask Inputs/MAIN.cloop_stat[60] <-> Status process data mapping/close_loop
//     PlcTask Inputs/MAIN.enable_stat[60] <-> Status process data mapping/enable
//     PlcTask Inputs/MAIN.force_rb_X[60] <-> Status process data mapping/force_rb_X
//     PlcTask Inputs/MAIN.force_rb_Y[60] <-> Status process data mapping/force_rb_Y
//     PlcTask Inputs/MAIN.force_rb_Z[60] <-> Status process data mapping/force_rb_Z
//     PlcTask Inputs/MAIN.force_sp_X[60] <-> Status process data mapping/force_sp_X
//     PlcTask Inputs/MAIN.force_sp_Y[60] <-> Status process data mapping/force_sp_Y
//     PlcTask Inputs/MAIN.force_sp_Z[60] <-> Status process data mapping/force_sp_Z
//     PlcTask Inputs/MAIN.pwm1[60] <-> Status process data mapping/pwm1
//     PlcTask Inputs/MAIN.pwm2[60] <-> Status process data mapping/pwm2
//     PlcTask Inputs/MAIN.pwm3[60] <-> Status process data mapping/pwm3
//     PlcTask Outputs/MAIN.enable_cmd[60] <-> Control process data mapping/enable
//     PlcTask Outputs/MAIN.force_cmd_X[60] <-> Control process data mapping/force_sp_X
//     PlcTask Outputs/MAIN.force_cmd_Y[60] <-> Control process data mapping/force_sp_Y
//     PlcTask Outputs/MAIN.force_cmd_Z[60] <-> Control process data mapping/force_sp_Z
//     PlcTask Outputs/MAIN.msthb[65] <-> Control process data mapping/msthb
//   SAsetGains/SAsetGains Instance <-> Device 1 (EtherCAT)/Box 63 (m1eph)/Box 66 (m1sa)
//     PlcTask Inputs/MAIN.cloop_stat[61] <-> Status process data mapping/close_loop
//     PlcTask Inputs/MAIN.enable_stat[61] <-> Status process data mapping/enable
//     PlcTask Inputs/MAIN.force_rb_X[61] <-> Status process data mapping/force_rb_X
//     PlcTask Inputs/MAIN.force_rb_Y[61] <-> Status process data mapping/force_rb_Y
//     PlcTask Inputs/MAIN.force_rb_Z[61] <-> Status process data mapping/force_rb_Z
//     PlcTask Inputs/MAIN.force_sp_X[61] <-> Status process data mapping/force_sp_X
//     PlcTask Inputs/MAIN.force_sp_Y[61] <-> Status process data mapping/force_sp_Y
//     PlcTask Inputs/MAIN.force_sp_Z[61] <-> Status process data mapping/force_sp_Z
//     PlcTask Inputs/MAIN.pwm1[61] <-> Status process data mapping/pwm1
//     PlcTask Inputs/MAIN.pwm2[61] <-> Status process data mapping/pwm2
//     PlcTask Inputs/MAIN.pwm3[61] <-> Status process data mapping/pwm3
//     PlcTask Outputs/MAIN.enable_cmd[61] <-> Control process data mapping/enable
//     PlcTask Outputs/MAIN.force_cmd_X[61] <-> Control process data mapping/force_sp_X
//     PlcTask Outputs/MAIN.force_cmd_Y[61] <-> Control process data mapping/force_sp_Y
//     PlcTask Outputs/MAIN.force_cmd_Z[61] <-> Control process data mapping/force_sp_Z
//     PlcTask Outputs/MAIN.msthb[66] <-> Control process data mapping/msthb
//   SAsetGains/SAsetGains Instance <-> Device 1 (EtherCAT)/Box 63 (m1eph)/Box 67 (m1sa)
//     PlcTask Inputs/MAIN.cloop_stat[62] <-> Status process data mapping/close_loop
//     PlcTask Inputs/MAIN.enable_stat[62] <-> Status process data mapping/enable
//     PlcTask Inputs/MAIN.force_rb_X[62] <-> Status process data mapping/force_rb_X
